# B&R Automation Studio project TD52 (part 150)

#### OpcMDE.st
```iecst
(*******************************************************************************
OPC_MDE	 Variables read or write to Measurement

This code is confidential AND proprietary to the INNIO Company.
It may NOT be used in any form, or reproduced in any manner, without the express
written permission of the INNIO Company.
Copyright, INNIO Company, 2022

- list addidtional customized IO channels

Customized modifications: -
------------------------

History:
-------
V1.00.0	09.12.2022		Vockenberger	Neu erstellt
V1.02.0	10.04.2024		Vockenberger	IN_DI.rP_Set auf IN_DI.rP_Act_FiltMDE + Mapping von MM2VIS.rP_Act_Filt
V1.03.0	05.03.2025		Vockenberger	added rOpcMDE_R[237] to rOpcMDE_R[300]

Instructions FOR use:
--------------------

Outstandings:
------------

*******************************************************************************)
PROGRAM _CYCLIC

	(*Connection OPC timeout*)
	(**BOOL**)
	TON_bComOpcBitMDE(IN:= bComOpcBitMDE, PT:=T#1s);
	IF TON_bComOpcBitMDE.Q THEN
		bOpcMDE_W[0] := FALSE;
	END_IF
	TON_bComOpcFailMDE(IN:= NOT bOpcMDE_W[0], PT:=T#1s);

	bComOpcBitMDE	:=	bOpcMDE_W[0];

	(*Abfrage welche Klopfüberwachung verwendet wird*)
	IF IN_DI.bKLS98_Active THEN
		rKnck_Sign[1] 	:= IN_DI.rKLS98_X_Window1[1];
		rKnck_Sign[2] 	:= IN_DI.rKLS98_X_Window1[2];
		rKnck_Sign[3] 	:= IN_DI.rKLS98_X_Window1[3];
		rKnck_Sign[4] 	:= IN_DI.rKLS98_X_Window1[4];
		rKnck_Sign[5] 	:= IN_DI.rKLS98_X_Window1[5];
		rKnck_Sign[6] 	:= IN_DI.rKLS98_X_Window1[6];
		rKnck_Sign[7] 	:= IN_DI.rKLS98_X_Window1[7];
		rKnck_Sign[8] 	:= IN_DI.rKLS98_X_Window1[8];
		rKnck_Sign[9] 	:= IN_DI.rKLS98_X_Window1[9];
		rKnck_Sign[10] 	:= IN_DI.rKLS98_X_Window1[10];
		rKnck_Sign[11] 	:= IN_DI.rKLS98_X_Window1[11];
		rKnck_Sign[12]	:= IN_DI.rKLS98_X_Window1[12];
		rKnck_Sign[13] 	:= IN_DI.rKLS98_X_Window1[13];
		rKnck_Sign[14] 	:= IN_DI.rKLS98_X_Window1[14];
		rKnck_Sign[15] 	:= IN_DI.rKLS98_X_Window1[15];
		rKnck_Sign[16] 	:= IN_DI.rKLS98_X_Window1[16];
		rKnck_Sign[17]	:= IN_DI.rKLS98_X_Window1[17];
		rKnck_Sign[18] 	:= IN_DI.rKLS98_X_Window1[18];
		rKnck_Sign[19] 	:= IN_DI.rKLS98_X_Window1[19];
		rKnck_Sign[20] 	:= IN_DI.rKLS98_X_Window1[20];
		rKnck_Sign[21] 	:= IN_DI.rKLS98_X_Window1[21];
		rKnck_Sign[22] 	:= IN_DI.rKLS98_X_Window1[22];
		rKnck_Sign[23] 	:= IN_DI.rKLS98_X_Window1[23];
		rKnck_Sign[24] 	:= IN_DI.rKLS98_X_Window1[24];
	ELSIF IN_DI.bSA_KLS_Active THEN
		rKnck_Sign[1] 	:= INT_TO_REAL(IN_DI.iU_SAFI_Win1[1]);
		rKnck_Sign[2] 	:= INT_TO_REAL(IN_DI.iU_SAFI_Win1[2]);
		rKnck_Sign[3] 	:= INT_TO_REAL(IN_DI.iU_SAFI_Win1[3]);
		rKnck_Sign[4] 	:= INT_TO_REAL(IN_DI.iU_SAFI_Win1[4]);
		rKnck_Sign[5] 	:= INT_TO_REAL(IN_DI.iU_SAFI_Win1[5]);
		rKnck_Sign[6] 	:= INT_TO_REAL(IN_DI.iU_SAFI_Win1[6]);
		rKnck_Sign[7] 	:= INT_TO_REAL(IN_DI.iU_SAFI_Win1[7]);
		rKnck_Sign[8] 	:= INT_TO_REAL(IN_DI.iU_SAFI_Win1[8]);
		rKnck_Sign[9] 	:= INT_TO_REAL(IN_DI.iU_SAFI_Win1[9]);
		rKnck_Sign[10] 	:= INT_TO_REAL(IN_DI.iU_SAFI_Win1[10]);
		rKnck_Sign[11] 	:= INT_TO_REAL(IN_DI.iU_SAFI_Win1[11]);
		rKnck_Sign[12]	:= INT_TO_REAL(IN_DI.iU_SAFI_Win1[12]);
		rKnck_Sign[13] 	:= INT_TO_REAL(IN_DI.iU_SAFI_Win1[13]);
		rKnck_Sign[14] 	:= INT_TO_REAL(IN_DI.iU_SAFI_Win1[14]);
		rKnck_Sign[15] 	:= INT_TO_REAL(IN_DI.iU_SAFI_Win1[15]);
		rKnck_Sign[16] 	:= INT_TO_REAL(IN_DI.iU_SAFI_Win1[16]);
		rKnck_Sign[17]	:= INT_TO_REAL(IN_DI.iU_SAFI_Win1[17]);
		rKnck_Sign[18] 	:= INT_TO_REAL(IN_DI.iU_SAFI_Win1[18]);
		rKnck_Sign[19] 	:= INT_TO_REAL(IN_DI.iU_SAFI_Win1[19]);
		rKnck_Sign[20] 	:= INT_TO_REAL(IN_DI.iU_SAFI_Win1[20]);
		rKnck_Sign[21] 	:= INT_TO_REAL(IN_DI.iU_SAFI_Win1[21]);
		rKnck_Sign[22] 	:= INT_TO_REAL(IN_DI.iU_SAFI_Win1[22]);
		rKnck_Sign[23] 	:= INT_TO_REAL(IN_DI.iU_SAFI_Win1[23]);
		rKnck_Sign[24] 	:= INT_TO_REAL(IN_DI.iU_SAFI_Win1[24]);
	ELSIF IN_DI.bSA_PI_Active THEN
		rKnck_Sign[1] 	:= IN_DI.rPr_Knck[1] * 1000;
		rKnck_Sign[2] 	:= IN_DI.rPr_Knck[2] * 1000;
		rKnck_Sign[3] 	:= IN_DI.rPr_Knck[3] * 1000;
		rKnck_Sign[4] 	:= IN_DI.rPr_Knck[4] * 1000;
		rKnck_Sign[5] 	:= IN_DI.rPr_Knck[5] * 1000;
		rKnck_Sign[6] 	:= IN_DI.rPr_Knck[6] * 1000;
		rKnck_Sign[7] 	:= IN_DI.rPr_Knck[7] * 1000;
		rKnck_Sign[8] 	:= IN_DI.rPr_Knck[8] * 1000;
		rKnck_Sign[9] 	:= IN_DI.rPr_Knck[9] * 1000;
		rKnck_Sign[10] 	:= IN_DI.rPr_Knck[10] * 1000;
		rKnck_Sign[11] 	:= IN_DI.rPr_Knck[11] * 1000;
		rKnck_Sign[12]	:= IN_DI.rPr_Knck[12] * 1000;
		rKnck_Sign[13] 	:= IN_DI.rPr_Knck[13] * 1000;
		rKnck_Sign[14] 	:= IN_DI.rPr_Knck[14] * 1000;
		rKnck_Sign[15] 	:= IN_DI.rPr_Knck[15] * 1000;
		rKnck_Sign[16] 	:= IN_DI.rPr_Knck[16] * 1000;
		rKnck_Sign[17]	:= IN_DI.rPr_Knck[17] * 1000;
		rKnck_Sign[18] 	:= IN_DI.rPr_Knck[18] * 1000;
		rKnck_Sign[19] 	:= IN_DI.rPr_Knck[19] * 1000;
		rKnck_Sign[20] 	:= IN_DI.rPr_Knck[20] * 1000;
		rKnck_Sign[21] 	:= IN_DI.rPr_Knck[21] * 1000;
		rKnck_Sign[22] 	:= IN_DI.rPr_Knck[22] * 1000;
		rKnck_Sign[23] 	:= IN_DI.rPr_Knck[23] * 1000;
		rKnck_Sign[24] 	:= IN_DI.rPr_Knck[24] * 1000;
	ELSE
		rKnck_Sign[1] 	:= 0;
		rKnck_Sign[2] 	:= 0;
		rKnck_Sign[3] 	:= 0;
		rKnck_Sign[4] 	:= 0;
		rKnck_Sign[5] 	:= 0;
		rKnck_Sign[6] 	:= 0;
		rKnck_Sign[7] 	:= 0;
		rKnck_Sign[8] 	:= 0;
		rKnck_Sign[9] 	:= 0;
		rKnck_Sign[10] 	:= 0;
		rKnck_Sign[11] 	:= 0;
		rKnck_Sign[12]	:= 0;
		rKnck_Sign[13] 	:= 0;
		rKnck_Sign[14] 	:= 0;
		rKnck_Sign[15] 	:= 0;
		rKnck_Sign[16] 	:= 0;
		rKnck_Sign[17]	:= 0;
		rKnck_Sign[18] 	:= 0;
		rKnck_Sign[19] 	:= 0;
		rKnck_Sign[20] 	:= 0;
		rKnck_Sign[21] 	:= 0;
		rKnck_Sign[22] 	:= 0;
		rKnck_Sign[23] 	:= 0;
		rKnck_Sign[24] 	:= 0;
	END_IF

	(*OPC Var to MDE*)
	rOpcMDE_R[0]	:=	DINT_TO_REAL(IN_DI.iCnt_OpHours);
	rOpcMDE_R[1]	:=	IN_DI.rT_EPU_EG[1];
	rOpcMDE_R[2]	:=	IN_DI.rT_EPU_EG[2];
	rOpcMDE_R[3]	:=	IN_DI.rT_EPU_EG[3];
	rOpcMDE_R[4]	:=	IN_DI.rT_EPU_EG[4];
	rOpcMDE_R[5]	:=	IN_DI.rT_EPU_EG[5];
	rOpcMDE_R[6]	:=	IN_DI.rT_EPU_EG[6];
	rOpcMDE_R[7]	:=	IN_DI.rT_EPU_EG[7];
	rOpcMDE_R[8]	:=	IN_DI.rT_EPU_EG[8];
	rOpcMDE_R[9]	:=	IN_DI.rT_EPU_EG[9];
	rOpcMDE_R[10]	:=	IN_DI.rT_EPU_EG[10];
	rOpcMDE_R[11]	:=	IN_DI.rT_EPU_EG[11];
	rOpcMDE_R[12]	:=	IN_DI.rT_EPU_EG[12];
	rOpcMDE_R[13]	:=	IN_DI.rT_EPU_EG[13];
	rOpcMDE_R[14]	:=	IN_DI.rT_EPU_EG[14];
	rOpcMDE_R[15]	:=	IN_DI.rT_EPU_EG[15];
	rOpcMDE_R[16]	:=	IN_DI.rT_EPU_EG[16];
	rOpcMDE_R[17]	:=	IN_DI.rT_EPU_EG[17];
	rOpcMDE_R[18]	:=	IN_DI.rT_EPU_EG[18];
	rOpcMDE_R[19]	:=	IN_DI.rT_EPU_EG[19];
	rOpcMDE_R[20]	:=	IN_DI.rT_EPU_EG[20];
	rOpcMDE_R[21]	:=	IN_DI.rT_EPU_EG[21];
	rOpcMDE_R[22]	:=	IN_DI.rT_EPU_EG[22];
	rOpcMDE_R[23]	:=	IN_DI.rT_EPU_EG[23];
	rOpcMDE_R[24]	:=	IN_DI.rT_EPU_EG[24];
	rOpcMDE_R[25]	:=	rKnck_Sign[1];
	rOpcMDE_R[26]	:=	rKnck_Sign[2];
	rOpcMDE_R[27]	:=	rKnck_Sign[3];
	rOpcMDE_R[28]	:=	rKnck_Sign[4];
	rOpcMDE_R[29]	:=	rKnck_Sign[5];
	rOpcMDE_R[30]	:=	rKnck_Sign[6];
	rOpcMDE_R[31]	:=	rKnck_Sign[7];
	rOpcMDE_R[32]	:=	rKnck_Sign[8];
	rOpcMDE_R[33]	:=	rKnck_Sign[9];
	rOpcMDE_R[34]	:=	rKnck_Sign[10];
	rOpcMDE_R[35]	:=	rKnck_Sign[11];
	rOpcMDE_R[36]	:=	rKnck_Sign[12];
	rOpcMDE_R[37]	:=	rKnck_Sign[13];
	rOpcMDE_R[38]	:=	rKnck_Sign[14];
	rOpcMDE_R[39]	:=	rKnck_Sign[15];
	rOpcMDE_R[40]	:=	rKnck_Sign[16];
	rOpcMDE_R[41]	:=	rKnck_Sign[17];
	rOpcMDE_R[42]	:=	rKnck_Sign[18];
	rOpcMDE_R[43]	:=	rKnck_Sign[19];
	rOpcMDE_R[44]	:=	rKnck_Sign[20];
	rOpcMDE_R[45]	:=	rKnck_Sign[21];
	rOpcMDE_R[46]	:=	rKnck_Sign[22];
	rOpcMDE_R[47]	:=	rKnck_Sign[23];
	rOpcMDE_R[48]	:=	rKnck_Sign[24];
	rOpcMDE_R[49]	:=	IN_DI.rCA_PI_Dur[1];
	rOpcMDE_R[50]	:=	IN_DI.rCA_PI_Dur[2];
	rOpcMDE_R[51]	:=	IN_DI.rCA_PI_Dur[3];
	rOpcMDE_R[52]	:=	IN_DI.rCA_PI_Dur[4];
	rOpcMDE_R[53]	:=	IN_DI.rCA_PI_Dur[5];
	rOpcMDE_R[54]	:=	IN_DI.rCA_PI_Dur[6];
	rOpcMDE_R[55]	:=	IN_DI.rCA_PI_Dur[7];
	rOpcMDE_R[56]	:=	IN_DI.rCA_PI_Dur[8];
	rOpcMDE_R[57]	:=	IN_DI.rCA_PI_Dur[9];
	rOpcMDE_R[58]	:=	IN_DI.rCA_PI_Dur[10];
	rOpcMDE_R[59]	:=	IN_DI.rCA_PI_Dur[11];
	rOpcMDE_R[60]	:=	IN_DI.rCA_PI_Dur[12];
	rOpcMDE_R[61]	:=	IN_DI.rCA_PI_Dur[13];
	rOpcMDE_R[62]	:=	IN_DI.rCA_PI_Dur[14];
	rOpcMDE_R[63]	:=	IN_DI.rCA_PI_Dur[15];
	rOpcMDE_R[64]	:=	IN_DI.rCA_PI_Dur[16];
	rOpcMDE_R[65]	:=	IN_DI.rCA_PI_Dur[17];
	rOpcMDE_R[66]	:=	IN_DI.rCA_PI_Dur[18];
	rOpcMDE_R[67]	:=	IN_DI.rCA_PI_Dur[19];
	rOpcMDE_R[68]	:=	IN_DI.rCA_PI_Dur[20];
	rOpcMDE_R[69]	:=	IN_DI.rCA_PI_Dur[21];
	rOpcMDE_R[70]	:=	IN_DI.rCA_PI_Dur[22];
	rOpcMDE_R[71]	:=	IN_DI.rCA_PI_Dur[23];
	rOpcMDE_R[72]	:=	IN_DI.rCA_PI_Dur[24];
	rOpcMDE_R[73]	:=	IN_DI.rCA_Ign_Act[1];
	rOpcMDE_R[74]	:=	IN_DI.rCA_Ign_Act[2];
	rOpcMDE_R[75]	:=	IN_DI.rCA_Ign_Act[3];
	rOpcMDE_R[76]	:=	IN_DI.rCA_Ign_Act[4];
	rOpcMDE_R[77]	:=	IN_DI.rCA_Ign_Act[5];
	rOpcMDE_R[78]	:=	IN_DI.rCA_Ign_Act[6];
	rOpcMDE_R[79]	:=	IN_DI.rCA_Ign_Act[7];
	rOpcMDE_R[80]	:=	IN_DI.rCA_Ign_Act[8];
	rOpcMDE_R[81]	:=	IN_DI.rCA_Ign_Act[9];
	rOpcMDE_R[82]	:=	IN_DI.rCA_Ign_Act[10];
	rOpcMDE_R[83]	:=	IN_DI.rCA_Ign_Act[11];
	rOpcMDE_R[84]	:=	IN_DI.rCA_Ign_Act[12];
	rOpcMDE_R[85]	:=	IN_DI.rCA_Ign_Act[13];
	rOpcMDE_R[86]	:=	IN_DI.rCA_Ign_Act[14];
	rOpcMDE_R[87]	:=	IN_DI.rCA_Ign_Act[15];
	rOpcMDE_R[88]	:=	IN_DI.rCA_Ign_Act[16];
	rOpcMDE_R[89]	:=	IN_DI.rCA_Ign_Act[17];
	rOpcMDE_R[90]	:=	IN_DI.rCA_Ign_Act[18];
	rOpcMDE_R[91]	:=	IN_DI.rCA_Ign_Act[19];
	rOpcMDE_R[92]	:=	IN_DI.rCA_Ign_Act[20];
	rOpcMDE_R[93]	:=	IN_DI.rCA_Ign_Act[21];
	rOpcMDE_R[94]	:=	IN_DI.rCA_Ign_Act[22];
	rOpcMDE_R[95]	:=	IN_DI.rCA_Ign_Act[23];
	rOpcMDE_R[96]	:=	IN_DI.rCA_Ign_Act[24];
	rOpcMDE_R[97]	:=	IN_DI.rU_Ign_Cyl[1];
	rOpcMDE_R[98]	:=	IN_DI.rU_Ign_Cyl[2];
	rOpcMDE_R[99]	:=	IN_DI.rU_Ign_Cyl[3];
	rOpcMDE_R[100]	:=	IN_DI.rU_Ign_Cyl[4];
	rOpcMDE_R[101]	:=	IN_DI.rU_Ign_Cyl[5];
	rOpcMDE_R[102]	:=	IN_DI.rU_Ign_Cyl[6];
	rOpcMDE_R[103]	:=	IN_DI.rU_Ign_Cyl[7];
	rOpcMDE_R[104]	:=	IN_DI.rU_Ign_Cyl[8];
	rOpcMDE_R[105]	:=	IN_DI.rU_Ign_Cyl[9];
	rOpcMDE_R[106]	:=	IN_DI.rU_Ign_Cyl[10];
	rOpcMDE_R[107]	:=	IN_DI.rU_Ign_Cyl[11];
	rOpcMDE_R[108]	:=	IN_DI.rU_Ign_Cyl[12];
	rOpcMDE_R[109]	:=	IN_DI.rU_Ign_Cyl[13];
	rOpcMDE_R[110]	:=	IN_DI.rU_Ign_Cyl[14];
	rOpcMDE_R[111]	:=	IN_DI.rU_Ign_Cyl[15];
	rOpcMDE_R[112]	:=	IN_DI.rU_Ign_Cyl[16];
	rOpcMDE_R[113]	:=	IN_DI.rU_Ign_Cyl[17];
	rOpcMDE_R[114]	:=	IN_DI.rU_Ign_Cyl[18];
	rOpcMDE_R[115]	:=	IN_DI.rU_Ign_Cyl[19];
	rOpcMDE_R[116]	:=	IN_DI.rU_Ign_Cyl[20];
	rOpcMDE_R[117]	:=	IN_DI.rU_Ign_Cyl[21];
	rOpcMDE_R[118]	:=	IN_DI.rU_Ign_Cyl[22];
	rOpcMDE_R[119]	:=	IN_DI.rU_Ign_Cyl[23];
	rOpcMDE_R[120]	:=	IN_DI.rU_Ign_Cyl[24];
	rOpcMDE_R[121]	:=	IN_DI.rT_CBearing[1];
	rOpcMDE_R[122]	:=	IN_DI.rT_CBearing[2];
	rOpcMDE_R[123]	:=	IN_DI.rT_CBearing[3];
	rOpcMDE_R[124]	:=	IN_DI.rT_CBearing[4];
	rOpcMDE_R[125]	:=	IN_DI.rT_CBearing[5];
	rOpcMDE_R[126]	:=	IN_DI.rT_CBearing[6];
	rOpcMDE_R[127]	:=	IN_DI.rT_CBearing[7];
	rOpcMDE_R[128]	:=	IN_DI.rT_CBearing[8];
	rOpcMDE_R[129]	:=	IN_DI.rT_CBearing[9];
	rOpcMDE_R[130]	:=	IN_DI.rT_CBearing[10];
	rOpcMDE_R[131]	:=	IN_DI.rT_CBearing[11];
	rOpcMDE_R[132]	:=	IN_DI.rT_CBearing[12];
	rOpcMDE_R[133]	:=	IN_DI.rT_CBearing[13];
	rOpcMDE_R[134]	:=	IN_DI.rT_CBearing[14];
	rOpcMDE_R[135]	:=	IN_DI.rT_CBearing[15];
	rOpcMDE_R[136]	:=	IN_DI.rT_CBearing[16];
	rOpcMDE_R[137]	:=	IN_DI.rT_CBearing[17];
	rOpcMDE_R[138]	:=	IN_DI.rT_CBearing[18];
	rOpcMDE_R[139]	:=	IN_DI.rT_CBearing[19];
	rOpcMDE_R[140]	:=	IN_DI.rT_CBearing[20];
	rOpcMDE_R[141]	:=	IN_DI.rT_CBearing[21];
	rOpcMDE_R[142]	:=	IN_DI.rT_CBearing[22];
	rOpcMDE_R[143]	:=	IN_DI.rT_CBearing[23];
	rOpcMDE_R[144]	:=	IN_DI.rT_CBearing[24];
	rOpcMDE_R[145]	:=	IN_DI.tT_MBearing[1].Ai;
	rOpcMDE_R[146]	:=	IN_DI.tT_MBearing[2].Ai;
	rOpcMDE_R[147]	:=	IN_DI.tT_MBearing[3].Ai;
	rOpcMDE_R[148]	:=	IN_DI.tT_MBearing[4].Ai;
	rOpcMDE_R[149]	:=	IN_DI.tT_MBearing[5].Ai;
	rOpcMDE_R[150]	:=	IN_DI.tT_MBearing[6].Ai;
	rOpcMDE_R[151]	:=	IN_DI.tT_MBearing[7].Ai;
	rOpcMDE_R[152]	:=	IN_DI.tT_MBearing[8].Ai;
	rOpcMDE_R[153]	:=	IN_DI.tT_MBearing[9].Ai;
	rOpcMDE_R[154]	:=	IN_DI.tT_MBearing[10].Ai;
	rOpcMDE_R[155]	:=	IN_DI.tT_MBearing[11].Ai;
	rOpcMDE_R[156]	:=	IN_DI.rCA_IgnP_Set;
	rOpcMDE_R[157]	:=	IN_DI.rCA_PI_Dur_Avg;
	rOpcMDE_R[158]	:=	IN_DI.rLam_Eng_LL_Set;
	rOpcMDE_R[159]	:=	IN_DI.rCA_Ign_Min;
	rOpcMDE_R[160]	:=	IN_DI.rCA_Ign_Max;
	rOpcMDE_R[161]	:=	IN_DI.rN_EngAct;
	IF IN_DI.tPos_Act_TV_A1.Exist THEN
		rOpcMDE_R[162]	:=	IN_DI.tPos_TV_A1.Ao;
	ELSE
		rOpcMDE_R[162]	:=	IN_DI.tPos_TV.Ao;
	END_IF
	rOpcMDE_R[163]	:=	IN_DI.rO2_NOxS_EngOut_B;
	rOpcMDE_R[164]	:=	IN_DI.tPos_TV_A2.Ao;
	rOpcMDE_R[165]	:=	IN_DI.tPos_TV_B1.Ao;
	rOpcMDE_R[166]	:=	IN_DI.tPos_TV_B2.Ao;
	IF IN_DI.bTSTC_Exist THEN
		rOpcMDE_R[167]	:=	IN_DI.tPos_CBV_A1.Ao;
		rOpcMDE_R[168]	:=	IN_DI.tPos_CBV_A2.Ao;
	ELSE
		rOpcMDE_R[167]	:=	IN_DI.tPos_CBV.Ao;
		rOpcMDE_R[168]	:=	IN_DI.tPos_CBV.Ao;
	END_IF
	rOpcMDE_R[169]	:=	IN_DI.rT_Ch_T2s_Avg;
	rOpcMDE_R[170]	:=	IN_DI.rCA_Ign_Avg;
	IF IN_DI.bTSTC_Exist THEN
		rOpcMDE_R[171]	:=	IN_DI.tPos_CBV_B1.Ao;
		rOpcMDE_R[172]	:=	IN_DI.tPos_CBV_B2.Ao;
	ELSE
		rOpcMDE_R[171]	:=	IN_DI.tPos_CBV34.Ao;
		rOpcMDE_R[172]	:=	IN_DI.tPos_CBV34.Ao;
	END_IF
	IF IN_DI.tPos_Act_TV_A1.Exist THEN
		rOpcMDE_R[173]	:=	IN_DI.tPos_Act_TV_A1.Ai;
	ELSE
		rOpcMDE_R[173]	:=	IN_DI.tPos_Act_TV.Ai;
	END_IF
	rOpcMDE_R[174]	:=	IN_DI.rO2_NOxS_EngOut;
	rOpcMDE_R[175]	:=	IN_DI.tPos_Act_TV_A2.Ai;
	rOpcMDE_R[176]	:=	IN_DI.tPos_Act_TV_B1.Ai;
	rOpcMDE_R[177]	:=	IN_DI.tPos_Act_TV_B2.Ai;
	IF IN_DI.tPos_Act_CBV_1.Exist THEN
		rOpcMDE_R[178]	:=	IN_DI.tPos_Act_CBV_1.Ai;
	ELSE
		rOpcMDE_R[178]	:=	IN_DI.tPos_Act_CBV_A1.Ai;
	END_IF
	IF IN_DI.tPos_Act_CBV_2.Exist THEN
		rOpcMDE_R[179]	:=	IN_DI.tPos_Act_CBV_2.Ai;
	ELSE
		rOpcMDE_R[179]	:=	IN_DI.tPos_Act_CBV_A2.Ai;
	END_IF
	IF IN_DI.tPos_Act_CBV_3.Exist THEN
		rOpcMDE_R[180]	:=	IN_DI.tPos_Act_CBV_3.Ai;
	ELSE
		rOpcMDE_R[180]	:=	IN_DI.tPos_Act_CBV_B1.Ai;
	END_IF
	rOpcMDE_R[181]	:=	IN_DI.tPos_Act_CBV_B2.Ai;
	rOpcMDE_R[182]	:=	UDINT_TO_REAL(IN_DI.ulGasFlowN[1]);
	rOpcMDE_R[183]	:=	UDINT_TO_REAL(IN_DI.ulGasFlowN[2]);
	rOpcMDE_R[184]	:=	UDINT_TO_REAL(IN_DI.ulGasFlowN[3]);
	rOpcMDE_R[185]	:=	IN_DI.rPr_EngLubOil;
	rOpcMDE_R[186]	:=	IN_DI.rT_EO;
	rOpcMDE_R[187]	:=	IN_DI.rT_ECW;
	rOpcMDE_R[188]	:=	IN_DI.rPr_ECW;
	rOpcMDE_R[189]	:=	IN_DI.rPr_TC_EOF_After;
	IF IN_DI.tPr_Ch_P2s_A.Exist THEN
		rOpcMDE_R[190]	:=	IN_DI.tPr_Ch_P2s_A.Ai;
	ELSE
		rOpcMDE_R[190]	:=	IN_DI.rPr_Ch_P2s;
	END_IF
	rOpcMDE_R[191]	:=	IN_DI.rO2_NOxS_EngOut_A;
	rOpcMDE_R[192]	:=	IN_DI.rPr_Ch_P2s_B;
	rOpcMDE_R[193]	:=	IN_DI.rPr_ECWaEng;
	rOpcMDE_R[194]	:=	IN_DI.rU_Avg_1;
	rOpcMDE_R[195]	:=	IN_DI.rI_Avg_1;
	rOpcMDE_R[196]	:=	IN_DI.rPF_Act_1;
	rOpcMDE_R[197]	:=	IN_DI.rPr_GR_I;
	rOpcMDE_R[198]	:=	IN_DI.rT_GR;
	rOpcMDE_R[199]	:=	IN_DI.rT_PCGT;
	rOpcMDE_R[200]	:=	IN_DI.rPr_PCG;
	rOpcMDE_R[201]	:=	IN_DI.rU_L1L2_1;
	rOpcMDE_R[202]	:=	IN_DI.rU_L2L3_1;
	rOpcMDE_R[203]	:=	IN_DI.rU_L3L1_1;
	rOpcMDE_R[204]	:=	IN_DI.rU_L1N_1;
	rOpcMDE_R[205]	:=	IN_DI.rU_L2N_1;
	rOpcMDE_R[206]	:=	IN_DI.rU_L3N_1;
	rOpcMDE_R[207]	:=	IN_DI.rPr_CC;
	rOpcMDE_R[208]	:=	IN_DI.rPr_EOF_DiffMon;
	rOpcMDE_R[209]	:=	IN_DI.rP_WorkAct_1;
	IF IN_DI.rNOx_NOxS_EngOut_Filt > 0.001 THEN
		rOpcMDE_R[210]	:=	IN_DI.rNOx_NOxS_EngOut_Filt;
	ELSE
		rOpcMDE_R[210]	:=	IN_DI.rNOx_NOxS_EngOut_A_Filt;
	END_IF
	rOpcMDE_R[211]	:=	IN_DI.rNOx_NOxS_EngOut_B_Filt;
	IF IN_DI.bN_TCHP_Exist THEN
		rOpcMDE_R[212]	:=	IN_DI.rN_TCHP;
	ELSE
		rOpcMDE_R[212]	:=	IN_DI.rN_TCHP_A;
	END_IF
	rOpcMDE_R[213]	:=	IN_DI.rN_TCHP_B;

	IF IN_DI.bN_TCHP_Exist THEN
		rOpcMDE_R[214]	:=	IN_DI.rN_TCLP;
	ELSE
		rOpcMDE_R[214]	:=	IN_DI.rN_TCLP_A;
	END_IF
	rOpcMDE_R[215]	:=	IN_DI.rN_TCLP_B;
	rOpcMDE_R[216]	:=	IN_DI.rGMU_Q_FuelGas[1];
	rOpcMDE_R[217]	:=	IN_DI.rGMU_Q_FuelGas[2];
	rOpcMDE_R[218]	:=	IN_DI.rGMU_Q_FuelGas[3];
	rOpcMDE_R[219]	:=	IN_DI.rGMU_Pos_Valve_Prom[1];
	rOpcMDE_R[220]	:=	IN_DI.rGMU_Pos_Valve_Prom[2];
	rOpcMDE_R[221]	:=	IN_DI.rGMU_Pos_Valve_Prom[3];
	rOpcMDE_R[222]	:=	IN_DI.rPr_PC_Diff;
	rOpcMDE_R[223]	:=	IN_DI.rOC_Consum_Avg;
	rOpcMDE_R[224]	:=	DINT_TO_REAL(IN_DI.iCnt_Starts);
	rOpcMDE_R[225]	:=	IN_DI.rP_Act_FiltMDE;
	rOpcMDE_R[226]	:=	IN_DI.rP_set_vis;
	rOpcMDE_R[227]	:=	IN_DI.rPr_EOaP;
	rOpcMDE_R[228]	:=	IN_DI.rT_Ch_T1LP;
	rOpcMDE_R[229]	:=	IN_DI.rPr_TC_EOF_Before;
	rOpcMDE_R[230]	:=	IN_DI.rPr_Ch_P2s_Avg;
	IF IN_DI.tPos_Act_WG.Exist THEN
		rOpcMDE_R[231]	:=	IN_DI.tPos_Act_WG.Ai;
		rOpcMDE_R[233]	:=	IN_DI.tPos_Set_WG.Ao;
	ELSE
		rOpcMDE_R[231]	:=	IN_DI.tPos_Act_WG_A.Ai;
		rOpcMDE_R[233]	:=	IN_DI.tPos_Set_WG_A.Ao;
	END_IF
	rOpcMDE_R[232]	:=	IN_DI.tPos_Act_WG_B.Ai;
	rOpcMDE_R[234]	:=	IN_DI.tPos_Set_WG_B.Ao;
	rOpcMDE_R[235]	:=	IN_DI.tT_ECWbEng.Ai;
	rOpcMDE_R[236]	:=	IN_DI.rT_Ch_T1HP_Avg;

	(*V1.03.0 Start*)
	rOpcMDE_R[237]	:=	IN_DI.rKnck_Intgr[1];
	rOpcMDE_R[238]	:=	IN_DI.rKnck_Intgr[2];
	rOpcMDE_R[239]	:=	IN_DI.rKnck_Intgr[3];
	rOpcMDE_R[240]	:=	IN_DI.rKnck_Intgr[4];
	rOpcMDE_R[241]	:=	IN_DI.rKnck_Intgr[5];
	rOpcMDE_R[242]	:=	IN_DI.rKnck_Intgr[6];
	rOpcMDE_R[243]	:=	IN_DI.rKnck_Intgr[7];
	rOpcMDE_R[244]	:=	IN_DI.rKnck_Intgr[8];
	rOpcMDE_R[245]	:=	IN_DI.rKnck_Intgr[9];
	rOpcMDE_R[246]	:=	IN_DI.rKnck_Intgr[10];
	rOpcMDE_R[247]	:=	IN_DI.rKnck_Intgr[11];
	rOpcMDE_R[248]	:=	IN_DI.rKnck_Intgr[12];
	rOpcMDE_R[249]	:=	IN_DI.rKnck_Intgr[13];
	rOpcMDE_R[250]	:=	IN_DI.rKnck_Intgr[14];
	rOpcMDE_R[251]	:=	IN_DI.rKnck_Intgr[15];
	rOpcMDE_R[252]	:=	IN_DI.rKnck_Intgr[16];
	rOpcMDE_R[253]	:=	IN_DI.rKnck_Intgr[17];
	rOpcMDE_R[254]	:=	IN_DI.rKnck_Intgr[18];
	rOpcMDE_R[255]	:=	IN_DI.rKnck_Intgr[19];
	rOpcMDE_R[256]	:=	IN_DI.rKnck_Intgr[20];
	rOpcMDE_R[257]	:=	IN_DI.rKnck_Intgr[21];
	rOpcMDE_R[258]	:=	IN_DI.rKnck_Intgr[22];
	rOpcMDE_R[259]	:=	IN_DI.rKnck_Intgr[23];
	rOpcMDE_R[260]	:=	IN_DI.rKnck_Intgr[24];
	rOpcMDE_R[261]	:=	IN_DI.rGen_T_In;
	rOpcMDE_R[262]	:=	IN_DI.rPr_Leanox_Dev;
	rOpcMDE_R[263]	:=	UINT_TO_REAL(usDurationPI_A);
	rOpcMDE_R[264]	:=	UINT_TO_REAL(usDurationPI_B);
	rOpcMDE_R[265]	:=	IN_DI.rPr_IMEP_Avg;
	rOpcMDE_R[266]	:=	IN_DI.rPr_CPP_Avg;
	rOpcMDE_R[267]	:=	IN_DI.rCA_MFBvar_Avg;
	rOpcMDE_R[268]	:=	IN_DI.rT_Ch_T2s_A;
	rOpcMDE_R[269]	:=	IN_DI.rT_Ch_T2s_B;
	rOpcMDE_R[270]	:=	IN_DI.rT_DAI;
	rOpcMDE_R[271]	:=	IN_DI.rPos_DAI_Set_A;
	rOpcMDE_R[272]	:=	IN_DI.rPos_DAI_Set_B;
	rOpcMDE_R[273]	:=	IN_DI.rPos_DAI_Act_A;
	rOpcMDE_R[274]	:=	IN_DI.rPos_DAI_Act_B;
	rOpcMDE_R[275]	:=	IN_DI.rFlow_Dem_DAI;
	rOpcMDE_R[276]	:=	IN_DI.rNOx_NOxS_CatOut_cor;
	rOpcMDE_R[277]	:=	IN_DI.rNOx_Em_AvgShortTerm;
	rOpcMDE_R[278]	:=	IN_DI.rFlow_SCR_UreaDosingOut;
	rOpcMDE_R[279]	:=	IN_DI.rT_SCR_UreaDosingUnit_Release;
	rOpcMDE_R[280]	:=	IN_DI.rNOx_Em_EngOut_mg_Set;
	rOpcMDE_R[281]	:=	IN_DI.rT_SCR_CatAvg;
	rOpcMDE_R[282]	:=	IN_DI.rO2_NOxS_CatOut;
	rOpcMDE_R[283]	:=	IN_DI.rHum_CatOut;
	rOpcMDE_R[284]	:=	IN_DI.rPr_GR_filt;
	rOpcMDE_R[285]	:=	IN_DI.rN_AirStarter;
	rOpcMDE_R[286]	:=	IN_DI.rBbBlower_y;
	rOpcMDE_R[287]	:=	IN_DI.rPr_MGT_a_Filt;
	rOpcMDE_R[288]	:=	IN_DI.rPr_PCGT_Out;
	rOpcMDE_R[289]	:=	IN_DI.rVol_Ch_Engine_Norm;
	rOpcMDE_R[290]	:=	IN_DI.rT_EG_LimMax;
	rOpcMDE_R[291]	:=	INT_TO_REAL(IN_DI.iNum_SkipCyl_Act);
	rOpcMDE_R[292]	:=	IN_DI.rFlow_OilSkid_DE;
	rOpcMDE_R[293]	:=	IN_DI.rFlow_OilSkid_NDE;
	rOpcMDE_R[294]	:=	IN_DI.tPIopenH[1].timing;
	rOpcMDE_R[295]	:=	IN_DI.rPr_AirStarter_Supply;
	rOpcMDE_R[296]	:=	IN_DI.rPos_AWG_Set_A;
	rOpcMDE_R[297]	:=	IN_DI.rPos_AWG_Set_B;
	rOpcMDE_R[298]	:=	IN_DI.rPos_AWG_Act_A;
	rOpcMDE_R[299]	:=	IN_DI.rPos_AWG_Act_B;
	rOpcMDE_R[300];
	(*V1.03.0 End*)

	rOpcMDE_R[301]	:=	IN_DI.rCust_ME[1];
	rOpcMDE_R[302]	:=	IN_DI.rCust_ME[2];
	rOpcMDE_R[303]	:=	IN_DI.rCust_ME[3];
	rOpcMDE_R[304]	:=	IN_DI.rCust_ME[4];
	rOpcMDE_R[305]	:=	IN_DI.rCust_ME[5];
	rOpcMDE_R[306]	:=	IN_DI.rCust_ME[6];
	rOpcMDE_R[307]	:=	IN_DI.rCust_ME[7];
	rOpcMDE_R[308]	:=	IN_DI.rCust_ME[8];
	rOpcMDE_R[309]	:=	IN_DI.rCust_ME[9];
	rOpcMDE_R[310]	:=	IN_DI.rCust_ME[10];
	rOpcMDE_R[311]	:=	IN_DI.rCust_ME[11];
	rOpcMDE_R[312]	:=	IN_DI.rCust_ME[12];
	rOpcMDE_R[313]	:=	IN_DI.rCust_ME[13];
	rOpcMDE_R[314]	:=	IN_DI.rCust_ME[14];
	rOpcMDE_R[315]	:=	IN_DI.rCust_ME[15];
	rOpcMDE_R[316]	:=	IN_DI.rCust_ME[16];
	rOpcMDE_R[317]	:=	IN_DI.rCust_ME[17];
	rOpcMDE_R[318]	:=	IN_DI.rCust_ME[18];
	rOpcMDE_R[319]	:=	IN_DI.rCust_ME[19];
	rOpcMDE_R[320]	:=	IN_DI.rCust_ME[20];
	rOpcMDE_R[321]	:=	IN_DI.rCust_ME[21];
	rOpcMDE_R[322]	:=	IN_DI.rCust_ME[22];
	rOpcMDE_R[323]	:=	IN_DI.rCust_ME[23];
	rOpcMDE_R[324]	:=	IN_DI.rCust_ME[24];
	rOpcMDE_R[325]	:=	IN_DI.rCust_ME[25];
	rOpcMDE_R[326]	:=	IN_DI.rCust_ME[26];
	rOpcMDE_R[327]	:=	IN_DI.rCust_ME[27];
	rOpcMDE_R[328]	:=	IN_DI.rCust_ME[28];
	rOpcMDE_R[329]	:=	IN_DI.rCust_ME[29];
	rOpcMDE_R[330]	:=	IN_DI.rCust_ME[30];
	rOpcMDE_R[331]	:=	IN_DI.rCust_ME[31];
	rOpcMDE_R[332]	:=	IN_DI.rCust_ME[32];
	rOpcMDE_R[333]	:=	IN_DI.rCust_ME[33];
	rOpcMDE_R[334]	:=	IN_DI.rCust_ME[34];
	rOpcMDE_R[335]	:=	IN_DI.rCust_ME[35];
	rOpcMDE_R[336]	:=	IN_DI.rCust_ME[36];
	rOpcMDE_R[337]	:=	IN_DI.rCust_ME[37];
	rOpcMDE_R[338]	:=	IN_DI.rCust_ME[38];
	rOpcMDE_R[339]	:=	IN_DI.rCust_ME[39];
	rOpcMDE_R[340]	:=	IN_DI.rCust_ME[40];
	rOpcMDE_R[341]	:=	IN_DI.rCust_ME[41];
	rOpcMDE_R[342]	:=	IN_DI.rCust_ME[42];
	rOpcMDE_R[343]	:=	IN_DI.rCust_ME[43];
	rOpcMDE_R[344]	:=	IN_DI.rCust_ME[44];
	rOpcMDE_R[345]	:=	IN_DI.rCust_ME[45];
	rOpcMDE_R[346]	:=	IN_DI.rCust_ME[46];
	rOpcMDE_R[347]	:=	IN_DI.rCust_ME[47];
	rOpcMDE_R[348]	:=	IN_DI.rCust_ME[48];
	rOpcMDE_R[349]	:=	IN_DI.rCust_ME[49];
	rOpcMDE_R[350]	:=	IN_DI.rCust_ME[50];
	rOpcMDE_R[351]	:=	IN_DI.rCust_ME[51];
	rOpcMDE_R[352]	:=	IN_DI.rCust_ME[52];
	rOpcMDE_R[353]	:=	IN_DI.rCust_ME[53];
	rOpcMDE_R[354]	:=	IN_DI.rCust_ME[54];
	rOpcMDE_R[355]	:=	IN_DI.rCust_ME[55];
	rOpcMDE_R[356]	:=	IN_DI.rCust_ME[56];
	rOpcMDE_R[357]	:=	IN_DI.rCust_ME[57];
	rOpcMDE_R[358]	:=	IN_DI.rCust_ME[58];
	rOpcMDE_R[359]	:=	IN_DI.rCust_ME[59];
	rOpcMDE_R[360]	:=	IN_DI.rCust_ME[60];
	rOpcMDE_R[361]	:=	IN_DI.rCust_ME[61];
	rOpcMDE_R[362]	:=	IN_DI.rCust_ME[62];
	rOpcMDE_R[363]	:=	IN_DI.rCust_ME[63];
	rOpcMDE_R[364]	:=	IN_DI.rCust_ME[64];
	rOpcMDE_R[365]	:=	IN_DI.rCust_ME[65];
	rOpcMDE_R[366]	:=	IN_DI.rCust_ME[66];
	rOpcMDE_R[367]	:=	IN_DI.rCust_ME[67];
	rOpcMDE_R[368]	:=	IN_DI.rCust_ME[68];
	rOpcMDE_R[369]	:=	IN_DI.rCust_ME[69];
	rOpcMDE_R[370]	:=	IN_DI.rCust_ME[70];
	rOpcMDE_R[371]	:=	IN_DI.rCust_ME[71];
	rOpcMDE_R[372]	:=	IN_DI.rCust_ME[72];
	rOpcMDE_R[373]	:=	IN_DI.rCust_ME[73];
	rOpcMDE_R[374]	:=	IN_DI.rCust_ME[74];
	rOpcMDE_R[375]	:=	IN_DI.rCust_ME[75];
	rOpcMDE_R[376]	:=	IN_DI.rCust_ME[76];
	rOpcMDE_R[377]	:=	IN_DI.rCust_ME[77];
	rOpcMDE_R[378]	:=	IN_DI.rCust_ME[78];
	rOpcMDE_R[379]	:=	IN_DI.rCust_ME[79];
	rOpcMDE_R[380]	:=	IN_DI.rCust_ME[80];
	rOpcMDE_R[381]	:=	IN_DI.rCust_ME[81];
	rOpcMDE_R[382]	:=	IN_DI.rCust_ME[82];
	rOpcMDE_R[383]	:=	IN_DI.rCust_ME[83];
	rOpcMDE_R[384]	:=	IN_DI.rCust_ME[84];
	rOpcMDE_R[385]	:=	IN_DI.rCust_ME[85];
	rOpcMDE_R[386]	:=	IN_DI.rCust_ME[86];
	rOpcMDE_R[387]	:=	IN_DI.rCust_ME[87];
	rOpcMDE_R[388]	:=	IN_DI.rCust_ME[88];
	rOpcMDE_R[389]	:=	IN_DI.rCust_ME[89];
	rOpcMDE_R[390]	:=	IN_DI.rCust_ME[90];
	rOpcMDE_R[391]	:=	IN_DI.rCust_ME[91];
	rOpcMDE_R[392]	:=	IN_DI.rCust_ME[92];
	rOpcMDE_R[393]	:=	IN_DI.rCust_ME[93];
	rOpcMDE_R[394]	:=	IN_DI.rCust_ME[94];
	rOpcMDE_R[395]	:=	IN_DI.rCust_ME[95];
	rOpcMDE_R[396]	:=	IN_DI.rCust_ME[96];
	rOpcMDE_R[397]	:=	IN_DI.rCust_ME[97];
	rOpcMDE_R[398]	:=	IN_DI.rCust_ME[98];
	rOpcMDE_R[399]	:=	IN_DI.rCust_ME[99];
	rOpcMDE_R[400]	:=	IN_DI.rCust_ME[100];
	rOpcMDE_R[401]	:=	IN_DI.rCust_ME[101];
	rOpcMDE_R[402]	:=	IN_DI.rCust_ME[102];
	rOpcMDE_R[403]	:=	IN_DI.rCust_ME[103];
	rOpcMDE_R[404]	:=	IN_DI.rCust_ME[104];
	rOpcMDE_R[405]	:=	IN_DI.rCust_ME[105];
	rOpcMDE_R[406]	:=	IN_DI.rCust_ME[106];
	rOpcMDE_R[407]	:=	IN_DI.rCust_ME[107];
	rOpcMDE_R[408]	:=	IN_DI.rCust_ME[108];
	rOpcMDE_R[409]	:=	IN_DI.rCust_ME[109];
	rOpcMDE_R[410]	:=	IN_DI.rCust_ME[110];
	rOpcMDE_R[411]	:=	IN_DI.rCust_ME[111];
	rOpcMDE_R[412]	:=	IN_DI.rCust_ME[112];
	rOpcMDE_R[413]	:=	IN_DI.rCust_ME[113];
	rOpcMDE_R[414]	:=	IN_DI.rCust_ME[114];
	rOpcMDE_R[415]	:=	IN_DI.rCust_ME[115];
	rOpcMDE_R[416]	:=	IN_DI.rCust_ME[116];
	rOpcMDE_R[417]	:=	IN_DI.rCust_ME[117];
	rOpcMDE_R[418]	:=	IN_DI.rCust_ME[118];
	rOpcMDE_R[419]	:=	IN_DI.rCust_ME[119];
	rOpcMDE_R[420]	:=	IN_DI.rCust_ME[120];

	rOpcMDE_R[421]	:=	IN_DI.rCust_ME_10ms[1];
	rOpcMDE_R[422]	:=	IN_DI.rCust_ME_10ms[2];
	rOpcMDE_R[423]	:=	IN_DI.rCust_ME_10ms[3];
	rOpcMDE_R[424]	:=	IN_DI.rCust_ME_10ms[4];
	rOpcMDE_R[425]	:=	IN_DI.rCust_ME_10ms[5];
	rOpcMDE_R[426]	:=	IN_DI.rCust_ME_10ms[6];
	rOpcMDE_R[427]	:=	IN_DI.rCust_ME_10ms[7];
	rOpcMDE_R[428]	:=	IN_DI.rCust_ME_10ms[8];
	rOpcMDE_R[429]	:=	IN_DI.rCust_ME_10ms[9];
	rOpcMDE_R[430]	:=	IN_DI.rCust_ME_10ms[10];
	rOpcMDE_R[431]	:=	IN_DI.rCust_ME_10ms[11];
	rOpcMDE_R[432]	:=	IN_DI.rCust_ME_10ms[12];
	rOpcMDE_R[433]	:=	IN_DI.rCust_ME_10ms[13];
	rOpcMDE_R[434]	:=	IN_DI.rCust_ME_10ms[14];
	rOpcMDE_R[435]	:=	IN_DI.rCust_ME_10ms[15];
	rOpcMDE_R[436]	:=	IN_DI.rCust_ME_10ms[16];
	rOpcMDE_R[437]	:=	IN_DI.rCust_ME_10ms[17];
	rOpcMDE_R[438]	:=	IN_DI.rCust_ME_10ms[18];
	rOpcMDE_R[439]	:=	IN_DI.rCust_ME_10ms[19];
	rOpcMDE_R[440]	:=	IN_DI.rCust_ME_10ms[20];

	bOpcMDE_R[0]	:=	IN_DI.bEOP1DC_Dem;
	(*V1.03.0 Start*)
	bOpcMDE_R[1]	:=	IN_DI.bEng_Start;
	bOpcMDE_R[2]	:=	IN_DI.bEng_Dem_Aut;
	bOpcMDE_R[3]	:=	IN_DI.bGCB_On;
	bOpcMDE_R[4]	:=	IN_DI.bAirST_ValEngage;
	bOpcMDE_R[5]	:=	IN_DI.bAirST_ValStart;
	bOpcMDE_R[6]	:=	IN_DI.bTCOV_CoClose;
	bOpcMDE_R[7]	:=	IN_DI.bScavVaFailure;
	bOpcMDE_R[8]	:=	IN_DI.bEng_Dem;
	bOpcMDE_R[9]	:=	IN_DI.bChargeOff_Dem;
	(*V1.03.0 End*)

	rOpcMDE_W;
	OUT_DI.rCust_From_PUMA[1]	:=	rOpcMDE_W[25];
	OUT_DI.rCust_From_PUMA[2]	:=	rOpcMDE_W[26];
	OUT_DI.rCust_From_PUMA[3]	:=	rOpcMDE_W[27];
	OUT_DI.rCust_From_PUMA[4]	:=	rOpcMDE_W[28];
	OUT_DI.rCust_From_PUMA[5]	:=	rOpcMDE_W[29];
	OUT_DI.rCust_From_PUMA[6]	:=	rOpcMDE_W[30];
	OUT_DI.rCust_From_PUMA[7]	:=	rOpcMDE_W[31];
	OUT_DI.rCust_From_PUMA[8]	:=	rOpcMDE_W[32];
	OUT_DI.rCust_From_PUMA[9]	:=	rOpcMDE_W[33];
	OUT_DI.rCust_From_PUMA[10]	:=	rOpcMDE_W[34];
	OUT_DI.rCust_From_PUMA[11]	:=	rOpcMDE_W[35];
	OUT_DI.rCust_From_PUMA[12]	:=	rOpcMDE_W[36];

	OUT_DI.rAMA_CH4_ppm		:=	rOpcMDE_W[41];
	OUT_DI.rAMA_THC_ppm		:=	rOpcMDE_W[42];
	OUT_DI.rAMA_CO_ppm		:=	rOpcMDE_W[43];
	OUT_DI.rAMA_CO2_per		:=	rOpcMDE_W[44];
	OUT_DI.rAMA_O2_per		:=	rOpcMDE_W[45];
	OUT_DI.rAMA_NO_ppm		:=	rOpcMDE_W[46];
	OUT_DI.rAMA_NOx_ppm		:=	rOpcMDE_W[47];
	OUT_DI.rAMA_Status		:=	rOpcMDE_W[48];
	rOpcMDE_W[49];
	rOpcMDE_W[50];

	bOpcMDE_W;

END_PROGRAM
```

#### OpcMDE.var
```iecst
VAR
	rKnck_Sign : ARRAY[0..24]OF REAL; (* Cylinder Knocking Value/Pressure *)
END_VAR
```

### Program Logical/DataInterface/IN_DI (IEC) - Var from Customiezd Modul

#### IN_DI.st
```iecst
(*******************************************************************************
IN_DI	Variables from other modules

This code is confidential AND proprietary to the INNIO Company.
It may NOT be used in any form, or reproduced in any manner, without the express
written permission of the INNIO Company.
Copyright, INNIO Company, 2022

- list addidtional customized IO channels

Customized modifications: -
------------------------

History:
-------
V1.01.0	31.07.2023		Vockenberger	Neu erstellt
		04.03.2024		Gruber St.		changed connection for gasvalves visualization
V1.01.1	19.03.2024		Gruber St.		changed connection for gas proportioning valves
										moved vis mixgas ratio to Gnl_GT
		27.03.2024		Gruber St. 		added H2-Sensor engine

Instructions FOR use:
--------------------

Outstandings:
------------

*******************************************************************************)
PROGRAM _CYCLIC

	(*Variablen die von anderen Modulen kommen*)
	IN_DI.rP_Act_Norm_Filt;
	MM2VIS.bBlocGasMixButton := IN_DI.bEng_Aux_Dem_CDR;
	MM2VIS.bPCG_GV_Open := IN_DI.bPCG_GV_Open;
	MM2VIS.bGV1_Open := IN_DI.bGV1_Open;
	MM2VIS.bGV2_Open := IN_DI.bGV2_Open; // AND MM2VIS.bDem_GV_PG AND NOT MM2VIS.bGV3_Open;
	MM2VIS.bGV3_Open := IN_DI.bGV3_Open; // AND MM2VIS.bDem_GV_SG AND NOT Para.bSG_MFC_Used AND NOT MM2VIS.bDem_GV_PG;
	MM2VIS.bEng_Run := IN_DI.bEng_Run;
	MM2VIS.rLam_Eng_LL_Set := IN_DI.rLam_Eng_LL_Set;
	MM2VIS.rGMU_Pos_Valve_Prom1 := IN_DI.rGMU_Pos_Valve_Prom[1];
	MM2VIS.rGMU_Pos_Valve_Prom2 := IN_DI.rGMU_Pos_Valve_Prom[2];
	MM2VIS.rGMU_Pos_Valve_Prom3 := IN_DI.rGMU_Pos_Valve_Prom[3];
	MM2VIS.iIdx_SelGasTyp	:= IN_DI.iIdx_SelGasTyp;
	MM2VIS.iIdx_Gtyp_Act	:= IN_DI.iIdx_Gtyp_Act;
	MM2VIS.rPr_Ch_P2s_Avg	:= IN_DI.rPr_Ch_P2s_Avg;
	MM2VIS.rCA_IgnP_Set	:=	IN_DI.rCA_IgnP_Set;
	MM2VIS.bGEN2_preM_Act	:=	IN_DI.bGEN2_preM_Act;
	MM2VIS.rGT_H2	:= IN_DI.rCust_ME[5] * 0.1;	// IN_DI.rGT_H2 * 100;
	MM2VIS.rCA_Ign_Avg		:=	IN_DI.rCA_Ign_Avg;
END_PROGRAM
```

### Program Logical/DataInterface/OUT_DI (IEC) - Var to Customiezd Modul

#### OUT_DI.st
```iecst
(*******************************************************************************
OUT_DI	Variables to other modules

This code is confidential AND proprietary to the INNIO Company.
It may NOT be used in any form, or reproduced in any manner, without the express
written permission of the INNIO Company.
Copyright, INNIO Company, 2022

- list addidtional customized IO channels

Customized modifications: -
------------------------

History:
-------
V1.00.0	14.09.2022		Vockenberger	Neu erstellt
V1.01.0 17.07.2023		Gruber St.		added setpoint for gasmixing with gas proportioning valve
		07.08.2023		Vockenberger	Ext Vorgaben von MDE/MyPlant
		04.03.2024		Gruber St.		added setpoints for admixing special gas with gas proportioning valve
V1.01.1 13.03.2024		Gruber St.		added variables for admixing H2

Instructions FOR use:
--------------------

Outstandings:
------------

*******************************************************************************)
PROGRAM _CYCLIC

	(*Aktivierung Vorwärmung, wenn Betriebswahlschalter auf aus ist *)
	IF EDGEPOS(MM2VIS.bPreHeatWDay_On) THEN	(*Aktivierung Vorwärmung vom Prüfstand über eine positiven Flanke*)
		VIS2MM.bECW_PreH_Dem_Customized := TRUE;
	ELSE
		VIS2MM.bECW_PreH_Dem_Customized := VIS2MM.bECW_PreH_Dem_Customized;
	END_IF

	OUT_DI.bECW_PreH_Dem_Customized := VIS2MM.bECW_PreH_Dem_Customized; (*Aktivierung Vorwärmung Prüfstandsseitig, wird im General_Di nochmal beschrieben*)

	(*Ext P-Vorgabe, kann über PUMA/MyPlant vorgegeben werden*)
	IF NOT MM2VIS.bMsg7000 AND VIS2MM.iSelExtP_OPC_Set = 1 THEN
		OUT_DI.bOPC_Dem := MM2VIS.bOPC_Dem;
		OUT_DI.rP_OPC_Set := MM2VIS.rP_OPC_Set;
	ELSIF VIS2MM.iSelExtP_OPC_Set = 2 THEN
		OUT_DI.rP_OPC_Set := MM2VIS.rP_OPC_Set;
		OUT_DI.bOPC_Dem := MM2VIS.bOPC_Dem;
	ELSE
		OUT_DI.rP_OPC_Set := 0.5;
		OUT_DI.bOPC_Dem := FALSE;
	END_IF
	OUT_DI.bBusAlive := MM2VIS.bBusAlive;

	(*Ext Vorgaben von MDE*)
	OUT_DI.rCA_IgnP_CylOffset			:= MM2VIS.rCA_IgnP_CylOffset;
	OUT_DI.bLeanox_Man_Cust				:= MM2VIS.bLeanox_Man_Cust;
	OUT_DI.rLam_Eng_LL_ManSet_Cust		:= MM2VIS.rLam_Eng_LL_ManSet_Cust;
	OUT_DI.rPr_Leanox_ManSet_Cust		:= MM2VIS.rPr_Leanox_ManSet_Cust;
	OUT_DI.bCA_IgnP_CylOffset_Active	:= MM2VIS.bCA_IgnP_CylOffset_Active;
	OUT_DI.bExtNOX_Active				:= MM2VIS.bExtNOX_Active;
	OUT_DI.rNOX_ManSet_Cust				:= MM2VIS.rNOX_ManSet_Cust;

	(*Gasmischen*)
	OUT_DI.bGT_CalibrateActive_Bus;
	OUT_DI.bCV_Bus_Active 		:= MM2VIS.bCV_Bus_Active;
	OUT_DI.rCV_Bus 				:= MM2VIS.rGT_CV_TB;
	OUT_DI.bOptGT_RatioMix_Set 	:= MM2VIS.bOptGT_RatioMix_Set;
	OUT_DI.rGT_RatioMix_Set		:= MM2VIS.rGT_RatioMix_Set;
	OUT_DI.bDem_GT3 			:= bDem_GT3;
	OUT_DI.rGT_RatioAdd			:= rGT_RatioAdd;
	OUT_DI.rH2_Set				:= rH2_Set;
	OUT_DI.rH2_Act_Calc			:= rH2_Act_Calc;
	OUT_DI.rH2_Act_Cube			:= rH2_Act_Cube;

END_PROGRAM
```

### Program Logical/DataInterface/PermDI (IEC, version 4.04.0) - + PermanentMemory

#### PermDICyclic.st - Cyclic code
```iecst
(*******************************************************************************
AGGR: read and write DIA.NE XT parameter to flash memory	(Cyclic)

This code is confidential and proprietary to the INNIO Jenbacher Company.
It may not be used in any form, or reproduced in any manner, without the express
written permission of the INNIO Company.
Copyright, INNIO Jenbacher Company, 2022

- every 10 seconds or at write once the parameter values are copied to the structure pm
- every 10 seconds the checksum of the parameter structure is calculate
- IF checksum has changed or write once is set the structure pm is written to
	the permanent memory data module

Customized modifications: -
------------------------

History:
-------
V1.00.0	16.09.2022	Vockenberger 	Neu erstellt
V1.01.0 07.08.2023	Vockenberger	im INIT Datenspeichergeändert, da neue Parameter dazukommen sind
V1.02.1 30.10.2024	Vockenberger	im INIT Datenspeichergeändert, da neue Parameter dazukommen sind

*******************************************************************************)
PROGRAM _CYCLIC

	(* 10 seconds timer *)
	TON_WritePMEM(IN := NOT TON_WritePMEM.Q, PT:= T#10s);
	TON_BlockMinFileAge(IN := bBlock_MinFileAge, PT:= T#10m);
	IF TON_BlockMinFileAge.Q  THEN bBlock_MinFileAge := FALSE; END_IF

	(* every 10 seconds or at write once the parameter values are copied to the structure pm *)
	IF TON_WritePMEM.Q OR write_once THEN

		(* ------------- V04.04.0 ---------------- *)   					(* permanent memory data *)
		pmm			:=	Para;						(* op.hours oxi cat *)

	END_IF;

	(* cyclic calcualtion of parameter checksum	*)
	IF TON_WritePMEM.Q THEN
		ulChecksum := 0;

		FOR ulPMPointer := ADR(pmm) TO (ADR(pmm) + pm_len - SIZEOF(ulChkValue)) DO
			memcpy(ADR(ulChkValue), ulPMPointer, SIZEOF(ulChkValue));
			ulChecksum := (ulChecksum XOR ulChkValue)+ulChkValue;
		END_FOR;

		IF ulChecksumOld <> ulChecksum THEN	(* if checksum has changed 		*)
			ulChecksumOld := ulChecksum;	(* save last cheksum value		*)
			bWriteDataObj := TRUE;			(* set flag for write checksum	*)
		END_IF;

	END_IF

	(* write structure pm to the permanent memory module *)
	IF ((bWriteDataObj AND NOT bBlock_MinFileAge) OR write_once) THEN

		DatObjWrite_01();									(* run data object write fub 				*)

		IF DatObjWrite_01.status <> ERR_FUB_BUSY THEN		(* wait if data object write fub is busy 	*)
			bWriteDataObj 	:= FALSE;						(* reset data object write flag				*)
			write_once 		:= FALSE;						(* reset write_once flag 					*)
			iPM_WriteCnt 	:= iPM_WriteCnt + 1;			(* counter for done data object module writes *)

			IF DatObjWrite_01.status = ERR_NOERROR THEN		(* if status = NO ERROR -> block further write requests for 10min to avoid CF wear down	*)
				bBlock_MinFileAge := TRUE;
			ELSE
				pm_Error := 2005;							(* set data object write error state		*)
			END_IF;
		END_IF;

	END_IF;

END_PROGRAM
```

#### PermDIInit.st - Initialization code
```iecst
(*******************************************************************************
AGGR: read and write DIA.NE XT parameter to flash memory	(init)

This code is confidential and proprietary to the INNIO Jenbacher Company.
It may not be used in any form, or reproduced in any manner, without the express
written permission of the INNIO Company.
Copyright, INNIO Jenbacher Company, 2022

- every 10 seconds or at write once the parameter values are copied to the structure pm
- every 10 seconds the checksum of the parameter structure is calculate
- IF checksum has changed or write once is set the structure pm is written to
	the permanent memory data module

Customized modifications: -
------------------------

History:
-------
V1.00.0	16.09.2022	Vockenberger 	Neu erstellt
V1.01.0 07.08.2023	Vockenberger	Datenspeichergeändert, da neue Parameter dazukommen sind
V1.01.1	20.03.2024	Gruber St.		Datenspeicher erhöht
V1.02.0 10.04.2024	Vockenberger	Datenspeichergeändert, da neue Parameter dazukommen sind
		23.04.2024	Gruber St.		Datenspeicher erhöht
V1.02.1 30.10.2024	Vockenberger	im INIT Datenspeichergeändert, da neue Parameter dazukommen sind

*******************************************************************************)

PROGRAM _INIT

	(* set some init parameters *)
	TON_WritePMEM(IN := FALSE, PT:= T#10s);			(* reset used timer function blocks 			*)

	pm_Error 	:= ERR_NOERROR;						(* reset permanent memory error	status			*)
	write_once 	:= FALSE;				 			(* reset flag for write permanent memory once	*)
	pm_len 		:= SIZEOF(pmm);						(* define data length of permenent memory		*)
	strcpy(ADR(ModulName),ADR('DataInterface::perm_DI'));	(* define name of permanent memory data module	*)

	(* check for existing permanent memory data module	*)
	DatObjInfo_01.enable:= TRUE;					(* enable FUB									*)
	DatObjInfo_01.pName := ADR(ModulName);			(* set permanent memory data module name 		*)
	DatObjInfo_01();								(* run data object info FUB						*)

	(* check error status of data object info FUB	*)
	IF DatObjInfo_01.status = ERR_NOERROR THEN		(* if no error	--> permanent memory data module exists	*)
		pm_id 	:= DatObjInfo_01.ident;				(* copy permanent memory data module ident			*)
		pm_p 	:= DatObjInfo_01.pDatObjMem;		(* copy permanent memory data module memory adres	*)
	ELSE
		bCreateDataObj := TRUE;						(* set flag for create new data object	*)
		pm_Error := 2001;							(* set permanent memory error status	*)
	END_IF;

	(* check length of parameter struct with length of data object *)

	CASE DatObjInfo_01.len OF

		1932: 		perm_par_vers  := 400;			(* 44 = length of perm_par V04.00.0 *)

			(* insert new perm_par Version here
			(* 		  bCreateDataObj := TRUE;		(* set flag for create new data object	*)
			(* xxxx:  perm_par_vers  := yyy;		(* xxxx = length of perm_par Vy.yy *)

		ELSE
		bCreateDataObj := TRUE;						(* set flag for create new data object	*)
	END_CASE;

	(* if permanent memory data module exist read data and copy to structure pm	*)
	IF pm_Error = ERR_NOERROR THEN					(* permanent memory data module exist 				*)
		DatObjRead_01.enable 		:= TRUE;		(* enable read permanent memory module data 		*)
		DatObjRead_01.ident 		:= pm_id;		(* set identifier of permanent memory data module	*)
		DatObjRead_01.Offset 		:= 0;			(* start at memory offest zero 						*)
		DatObjRead_01.pDestination := ADR(pmm);		(* set permanent data destination adress			*)
		DatObjRead_01.len 			:= DatObjInfo_01.len;	(* set length of permanent data module		*)

		REPEAT	(* repeat until data of permanent memory data module have been read *)
			DatObjRead_01();						(* FUB read data from permanent data module 		*)
			UNTIL	DatObjRead_01.status <> ERR_FUB_BUSY		(* wait if FUB is busy 	*)
		END_REPEAT;

		IF DatObjRead_01.status <> ERR_NOERROR THEN	(* if status of read permanent data moduel is not OK 	*)
			pm_Error :=2002;						(* set permanent memory error status					*)
		END_IF
	END_IF;

	IF NOT bCreateDataObj THEN
		(* if permanent memory data module exist read data and copy to structure pm	*)
		IF pm_Error = ERR_NOERROR THEN					(* permanent memory data module exist 				*)
			DatObjRead_01.enable 		:= TRUE;		(* enable read permanent memory module data 		*)
			DatObjRead_01.ident 		:= pm_id;		(* set identifier of permanent memory data module	*)
			DatObjRead_01.Offset 		:= 0;			(* start at memory offest zero 						*)
			DatObjRead_01.pDestination := ADR(pmm);		(* set permanent data destination adress			*)
			DatObjRead_01.len 			:= DatObjInfo_01.len;	(* set length of permanent data module		*)

			REPEAT	(* repeat until data of permanent memory data module have been read *)
				DatObjRead_01();						(* FUB read data from permanent data module 		*)
				UNTIL	DatObjRead_01.status <> ERR_FUB_BUSY		(* wait if FUB is busy 	*)
			END_REPEAT;

			IF DatObjRead_01.status <> ERR_NOERROR THEN	(* if status of read permanent data moduel is not OK 	*)
				pm_Error :=2012;						(* set permanent memory error status					*)
			END_IF
		END_IF;

		(* if permanent memory data module exist --> copy data from structure pm to program parameter *)
		IF pm_Error = ERR_NOERROR THEN

			(************ Permanent structure ************)
			(* ------------- V04.04.0 ---------------- *)		(* permanent memory data *)
			Para				:=	pmm;

		END_IF;
	END_IF

	(* create new permanent memory data module	*)
	IF bCreateDataObj THEN

		(* try to delete old data module *)
		DatObjDelete_PermMem.enable := TRUE;
		DatObjDelete_PermMem.ident 	:= pm_id;

		REPEAT	(* repeat until delete of permanent memory data module is ready *)
			DatObjDelete_PermMem();		(* FUB for delete permanent memory data module *)
			UNTIL	DatObjDelete_PermMem.status <> ERR_FUB_BUSY		(* wait if FUB is busy 	*)
		END_REPEAT;

		(* create new one *)
		DatObjCreate_01.enable	 := TRUE;			(* enable create permanent memory data module FUB 	*)
		DatObjCreate_01.grp 	 := 0;				(* must to be set to zero							*)
		DatObjCreate_01.pName 	 := ADR(ModulName);	(* set permanent memory data module name 			*)
		DatObjCreate_01.len 	 := pm_len;			(* set length ofpermanent memory data module		*)
		DatObjCreate_01.MemType  := doUSRROM;		(* create permanent memory data module at USERROM	*)
		DatObjCreate_01.Option 	 := 0;				(* cyclic checksum monitoring is on					*)
		DatObjCreate_01.pCpyData := 0;				(* no data will be copied do the permanent memory data module *)

		pm_Error:= 2003;							(* set permanent memory error status	*)

		REPEAT	(* repeat until generation of permanent memory data module is ready *)
			DatObjCreate_01();						(* FUB for create permanent memory data module 		*)
			UNTIL	DatObjCreate_01.status <> ERR_FUB_BUSY		(* wait if FUB is busy 	*)
		END_REPEAT;

		IF DatObjCreate_01.status = ERR_NOERROR THEN	(* is creation of permanent memory data module OK 	*)
			pm_p 	:= DatObjCreate_01.pDatObjMem;		(* set memory adress of permanent memory data module*)
			pm_id 	:= DatObjCreate_01.ident;			(* set identifier of permanent memory data module 	*)
		ELSE
			pm_Error:= 2004;							(* set permanent memory error status	*)
		END_IF;
	END_IF;

	(* prepare parameter for permanent memory data write in cyclic task *)
	IF pm_Error < 2004 THEN							(* permanent memory data module exist or has been created	*)
		DatObjWrite_01.enable 	:= TRUE;			(* enable permanent memory data module read FUB 	*)
		DatObjWrite_01.ident 	:= pm_id;			(* set identifier of permanent memory data module 	*)
		DatObjWrite_01.Offset 	:= 0;				(* start at memory offest zero 						*)
		DatObjWrite_01.pSource 	:= ADR(pmm);			(* set permanent memory data module name 			*)
		DatObjWrite_01.len 		:= pm_len;			(* set length ofpermanent memory data module		*)
	END_IF;

	(* calcualte actual checksum of parameter structure	*)
	ulChecksumOld := 0;			(* reset checksum value *)

	FOR ulPMPointer := ADR(pmm) TO (ADR(pmm) + pm_len - SIZEOF(ulChkValue)) DO
		memcpy(ADR(ulChkValue), ulPMPointer, SIZEOF(ulChkValue));
		ulChecksumOld := ulChecksumOld XOR ulChkValue;
	END_FOR;

END_PROGRAM
```

#### PermDI.var - Local variables
```iecst
VAR
	pm_Error : UINT;
	write_once : BOOL;
	pm_len : UDINT;
	ModulName : STRING[35];
	DatObjInfo_01 : DatObjInfo;
	pm_id : UDINT;
	pm_p : UDINT;
	bCreateDataObj : BOOL;
	perm_par_vers : UINT;
	DatObjRead_01 : DatObjRead;
	DatObjDelete_PermMem : DatObjDelete;
	DatObjCreate_01 : DatObjCreate;
	DatObjWrite_01 : DatObjWrite;
	ulChecksumOld : UDINT;
	ulPMPointer : UDINT;
	ulChkValue : UDINT;
	TON_WritePMEM : TON;
	ulChecksum : UDINT;
	bWriteDataObj : BOOL;
	TON_BlockMinFileAge : TON; (*waiting time without file write after successful performed write*)
	bBlock_MinFileAge : BOOL := FALSE; (*pause the perm file write after each sucessful write*)
	iPM_WriteCnt : UDINT; (* *) (*old VarName: usPMWriteCnt*)
END_VAR
VAR CONSTANT
	ERR_NOERROR : UINT := 0;
END_VAR
VAR
	pmm : Perm_DI_struct;
END_VAR
```

### Program Logical/DataInterface/VIS2PermDI (IEC, version 4.04.0) - + PermanentMemory

#### VIS2PermDICyclic.st - Cyclic code
```iecst
(*******************************************************************************
AGGR: read and write DIA.NE XT parameter to flash memory	(Cyclic)

This code is confidential and proprietary to the INNIO Jenbacher Company.
It may not be used in any form, or reproduced in any manner, without the express
written permission of the INNIO Company.
Copyright, INNIO Jenbacher Company, 2022

- every 10 seconds or at write once the parameter values are copied to the structure pm
- every 10 seconds the checksum of the parameter structure is calculate
- IF checksum has changed or write once is set the structure pm is written to
	the permanent memory data module

Customized modifications: -
------------------------

History:
-------
V1.00.0	16.09.2022	Vockenberger 	Neu erstellt
V1.03.0	22.01.2025	Gruber St.		added rCustEng2TB

*******************************************************************************)
PROGRAM _CYCLIC

	(* 10 seconds timer *)
	TON_WritePMEM(IN := NOT TON_WritePMEM.Q, PT:= T#10s);
	TON_BlockMinFileAge(IN := bBlock_MinFileAge, PT:= T#10m);
	IF TON_BlockMinFileAge.Q  THEN bBlock_MinFileAge := FALSE; END_IF

	(* every 10 seconds or at write once the parameter values are copied to the structure pm *)
	IF TON_WritePMEM.Q OR write_once THEN

		(* ------------- V04.04.0 ---------------- *)   					(* permanent memory data *)
		VIS2pmm.rFC_ChCW_LT_PuSet		:=	VIS2MM.rFC_ChCW_LT_PuSet;
		VIS2pmm.rFC_ChCW_HT_PuSet		:=	VIS2MM.rFC_ChCW_HT_PuSet;
		VIS2pmm.rFC_ChCW_LT_LP_PuSet	:=	VIS2MM.rFC_ChCW_LT_LP_PuSet;
		VIS2pmm.rFC_ChCW_LT_HP_PuSet	:=	VIS2MM.rFC_ChCW_LT_HP_PuSet;
		VIS2pmm.rFC_ChCW_HT_LP_PuSet	:=	VIS2MM.rFC_ChCW_HT_LP_PuSet;
		VIS2pmm.rFC_ChCW_HT_HP_PuSet	:=	VIS2MM.rFC_ChCW_HT_HP_PuSet;
		VIS2pmm.rFC_ECW_PuSet			:=	VIS2MM.rFC_ECW_PuSet;
		VIS2pmm.rFC_OCW_PuSet			:=	VIS2MM.rFC_OCW_PuSet;
		VIS2pmm.rCtr_RW_CV_Set			:=	VIS2MM.rCtr_RW_CV_Set;
		VIS2pmm.rCtr_RW_HE_Set			:=	VIS2MM.rCtr_RW_HE_Set;
		VIS2pmm.rCtr_RW_LT_1_Set		:=	VIS2MM.rCtr_RW_LT_1_Set;
		VIS2pmm.rCtr_RW_HT_1_Set		:=	VIS2MM.rCtr_RW_HT_1_Set;
		VIS2pmm.rCtr_RW_LT_2_Set		:=	VIS2MM.rCtr_RW_LT_2_Set;
		VIS2pmm.rCtr_RW_HT_2_Set		:=	VIS2MM.rCtr_RW_HT_2_Set;
		VIS2pmm.rCtr_RW_ECW_1_Set		:=	VIS2MM.rCtr_RW_ECW_1_Set;
		VIS2pmm.rCtr_RW_OCW_1_Set		:=	VIS2MM.rCtr_RW_OCW_1_Set;
		VIS2pmm.rCtr_RW_ECW_2_Set		:=	VIS2MM.rCtr_RW_ECW_2_Set;
		VIS2pmm.rCtr_RW_OCW_2_Set		:=	VIS2MM.rCtr_RW_OCW_2_Set;
		VIS2pmm.rMan_SRC_ByFlap_Set		:=	VIS2MM.rMan_SRC_ByFlap_Set;
		VIS2pmm.bECW_PreH_Dem_Customized := VIS2MM.bECW_PreH_Dem_Customized;
		VIS2pmm.rCtr_ChCW_LT_In_Y_set 	:=	VIS2MM.tCtr_ChCW_LT_In.Y_set;
		VIS2pmm.rCtr_ChCW_HT_In_Y_set 	:=	VIS2MM.tCtr_ChCW_HT_In.Y_set;
		VIS2pmm.rCtr_ChCW_LT_In_Y_set 	:=	VIS2MM.tCtr_ChCW_LT_In.Y_set;
		VIS2pmm.rCtr_ChCW_LT_In_Y_set 	:=	VIS2MM.tCtr_ChCW_LT_In.Y_set;
		VIS2pmm.rCtr_ChCW_HT_In_Y_set 	:=	VIS2MM.tCtr_ChCW_HT_In.Y_set;
		VIS2pmm.rCtr_ChCW_HT_In_Y_set 	:=	VIS2MM.tCtr_ChCW_HT_In.Y_set;
		VIS2pmm.rCtr_ECW_In_Y_set 		:=	VIS2MM.tCtr_ECW_In.Y_set;
		VIS2pmm.rCtr_OCW_In_Y_set 		:=	VIS2MM.tCtr_OCW_In.Y_set;
		VIS2pmm.bCtr_ChCW_LT_In_Y_set_Active := VIS2MM.tCtr_ChCW_LT_In.Y_set_Active;
		VIS2pmm.bCtr_ChCW_HT_In_Y_set_Active := VIS2MM.tCtr_ChCW_HT_In.Y_set_Active;
		VIS2pmm.bCtr_ChCW_LT_LP_In_Y_set_Active := VIS2MM.tCtr_ChCW_LT_LP_In.Y_set_Active;
		VIS2pmm.bCtr_ChCW_LT_HP_In_Y_set_Active := VIS2MM.tCtr_ChCW_LT_HP_In.Y_set_Active;
		VIS2pmm.bCtr_ChCW_HT_LP_In_Y_set_Active := VIS2MM.tCtr_ChCW_HT_LP_In.Y_set_Active;
		VIS2pmm.bCtr_ChCW_HT_HP_In_Y_set_Active := VIS2MM.tCtr_ChCW_HT_HP_In.Y_set_Active;
		VIS2pmm.bCtr_ECW_In_Y_set_Active 	:= VIS2MM.tCtr_ECW_In.Y_set_Active;
		VIS2pmm.bCtr_OCW_In_Y_set_Active 	:= VIS2MM.tCtr_OCW_In.Y_set_Active;
		VIS2pmm.bDem_ERV_Aut_Vis			:= VIS2MM.bDem_ERV_Aut_Vis;
		VIS2pmm.rMan_EG_Flap_Set			:= VIS2MM.rMan_EG_Flap_Set;
		VIS2pmm.rCust_Eng2TB				:= VIS2MM.rCust_Eng2TB;
		VIS2pmm.tPreHeatWDayLT				:= VIS2MM.tPreHeatWDayLT;
		VIS2pmm.bPreHeatWDayLT_CtrActive	:= VIS2MM.bPreHeatWDayLT_CtrActive;
		VIS2pmm.bLT_PreH_Dem				:= VIS2MM.bLT_PreH_Dem;
		VIS2pmm.rT_LT_HP_Preh				:= VIS2MM.rT_LT_HP_Preh;
		VIS2pmm.rT_LT_LP_Preh				:= VIS2MM.rT_LT_LP_Preh;
		VIS2pmm.bSel_PG_Comp				:= VIS2MM.bSel_PG_Comp;
		VIS2pmm.bSel_PG_TraceHeat			:= VIS2MM.bSel_PG_TraceHeat;
		VIS2pmm.bSel_PG_TraceHeat_TimeCtr	:= VIS2MM.bSel_PG_TraceHeat_TimeCtr;
		VIS2pmm.rCtr_PG_CompSet				:= VIS2MM.rCtr_PG_CompSet;
		VIS2pmm.rOp_ExhFlap					:= VIS2MM.rOp_ExhFlap;
		VIS2pmm.bCool_Air_Active			:= VIS2MM.bCool_Air_Active;
	END_IF;

	(* cyclic calcualtion of parameter checksum	*)
	IF TON_WritePMEM.Q THEN
		ulChecksum := 0;

		FOR ulPMPointer := ADR(VIS2pmm) TO (ADR(VIS2pmm) + pm_len - SIZEOF(ulChkValue)) DO
			memcpy(ADR(ulChkValue), ulPMPointer, SIZEOF(ulChkValue));
			ulChecksum := (ulChecksum XOR ulChkValue)+ulChkValue;
		END_FOR;

		IF ulChecksumOld <> ulChecksum THEN	(* if checksum has changed 		*)
			ulChecksumOld := ulChecksum;	(* save last cheksum value		*)
			bWriteDataObj := TRUE;			(* set flag for write checksum	*)
		END_IF;

	END_IF

	(* write structure pm to the permanent memory module *)
	IF ((bWriteDataObj AND NOT bBlock_MinFileAge) OR write_once) THEN

		DatObjWrite_01();									(* run data object write fub 				*)

		IF DatObjWrite_01.status <> ERR_FUB_BUSY THEN		(* wait if data object write fub is busy 	*)
			bWriteDataObj 	:= FALSE;						(* reset data object write flag				*)
			write_once 		:= FALSE;						(* reset write_once flag 					*)
			iPM_WriteCnt 	:= iPM_WriteCnt + 1;			(* counter for done data object module writes *)

			IF DatObjWrite_01.status = ERR_NOERROR THEN		(* if status = NO ERROR -> block further write requests for 10min to avoid CF wear down	*)
				bBlock_MinFileAge := TRUE;
			ELSE
				pm_Error := 2005;							(* set data object write error state		*)
			END_IF;
		END_IF;

	END_IF;

END_PROGRAM
```

#### VIS2PermDIInit.st - Initialization code
```iecst
(*******************************************************************************
AGGR: read and write DIA.NE XT parameter to flash memory	(init)

This code is confidential and proprietary to the INNIO Jenbacher Company.
It may not be used in any form, or reproduced in any manner, without the express
written permission of the INNIO Company.
Copyright, INNIO Jenbacher Company, 2022

- every 10 seconds or at write once the parameter values are copied to the structure pm
- every 10 seconds the checksum of the parameter structure is calculate
- IF checksum has changed or write once is set the structure pm is written to
	the permanent memory data module

Customized modifications: -
------------------------

History:
-------
V1.00.0	16.09.2022	Vockenberger 	Neu erstellt
V1.03.0	22.01.2025	Gruber St.		added rCustEng2TB

*******************************************************************************)

PROGRAM _INIT

	(* set some init parameters *)
	TON_WritePMEM(IN := FALSE, PT:= T#10s);			(* reset used timer function blocks 			*)

	pm_Error 	:= ERR_NOERROR;						(* reset permanent memory error	status			*)
	write_once 	:= FALSE;				 			(* reset flag for write permanent memory once	*)
	pm_len 		:= SIZEOF(VIS2pmm);						(* define data length of permenent memory		*)
	strcpy(ADR(ModulName),ADR('DataInterface::VISpm_DI'));	(* define name of permanent memory data module	*)

	(* check for existing permanent memory data module	*)
	DatObjInfo_01.enable:= TRUE;					(* enable FUB									*)
	DatObjInfo_01.pName := ADR(ModulName);			(* set permanent memory data module name 		*)
	DatObjInfo_01();								(* run data object info FUB						*)

	(* check error status of data object info FUB	*)
	IF DatObjInfo_01.status = ERR_NOERROR THEN		(* if no error	--> permanent memory data module exists	*)
		pm_id 	:= DatObjInfo_01.ident;				(* copy permanent memory data module ident			*)
		pm_p 	:= DatObjInfo_01.pDatObjMem;		(* copy permanent memory data module memory adres	*)
	ELSE
		bCreateDataObj := TRUE;						(* set flag for create new data object	*)
		pm_Error := 2001;							(* set permanent memory error status	*)
	END_IF;

	(* check length of parameter struct with length of data object *)

	CASE DatObjInfo_01.len OF

		456: 		perm_par_vers  := 400;			(* 44 = length of perm_par V04.00.0 *)

			(* insert new perm_par Version here
			(* 		  bCreateDataObj := TRUE;		(* set flag for create new data object	*)
			(* xxxx:  perm_par_vers  := yyy;		(* xxxx = length of perm_par Vy.yy *)

		ELSE
		bCreateDataObj := TRUE;						(* set flag for create new data object	*)
	END_CASE;

	(* if permanent memory data module exist read data and copy to structure pm	*)
	IF pm_Error = ERR_NOERROR THEN					(* permanent memory data module exist 				*)
		DatObjRead_01.enable 		:= TRUE;		(* enable read permanent memory module data 		*)
		DatObjRead_01.ident 		:= pm_id;		(* set identifier of permanent memory data module	*)
		DatObjRead_01.Offset 		:= 0;			(* start at memory offest zero 						*)
		DatObjRead_01.pDestination := ADR(VIS2pmm);		(* set permanent data destination adress			*)
		DatObjRead_01.len 			:= DatObjInfo_01.len;	(* set length of permanent data module		*)

		REPEAT	(* repeat until data of permanent memory data module have been read *)
			DatObjRead_01();						(* FUB read data from permanent data module 		*)
			UNTIL	DatObjRead_01.status <> ERR_FUB_BUSY		(* wait if FUB is busy 	*)
		END_REPEAT;

		IF DatObjRead_01.status <> ERR_NOERROR THEN	(* if status of read permanent data moduel is not OK 	*)
			pm_Error :=2002;						(* set permanent memory error status					*)
		END_IF
	END_IF;

	IF NOT bCreateDataObj THEN
		(* if permanent memory data module exist read data and copy to structure pm	*)
		IF pm_Error = ERR_NOERROR THEN					(* permanent memory data module exist 				*)
			DatObjRead_01.enable 		:= TRUE;		(* enable read permanent memory module data 		*)
			DatObjRead_01.ident 		:= pm_id;		(* set identifier of permanent memory data module	*)
			DatObjRead_01.Offset 		:= 0;			(* start at memory offest zero 						*)
			DatObjRead_01.pDestination := ADR(VIS2pmm);		(* set permanent data destination adress			*)
			DatObjRead_01.len 			:= DatObjInfo_01.len;	(* set length of permanent data module		*)

			REPEAT	(* repeat until data of permanent memory data module have been read *)
				DatObjRead_01();						(* FUB read data from permanent data module 		*)
				UNTIL	DatObjRead_01.status <> ERR_FUB_BUSY		(* wait if FUB is busy 	*)
			END_REPEAT;

			IF DatObjRead_01.status <> ERR_NOERROR THEN	(* if status of read permanent data moduel is not OK 	*)
				pm_Error :=2012;						(* set permanent memory error status					*)
			END_IF
		END_IF;

		(* if permanent memory data module exist --> copy data from structure pm to program parameter *)
		IF pm_Error = ERR_NOERROR THEN

			(************ Permanent structure ************)
			(* ------------- V04.04.0 ---------------- *)		(* permanent memory data *)
			VIS2MM.rFC_ChCW_LT_PuSet		:=	VIS2pmm.rFC_ChCW_LT_PuSet;
			VIS2MM.rFC_ChCW_HT_PuSet		:=	VIS2pmm.rFC_ChCW_HT_PuSet;
			VIS2MM.rFC_ChCW_LT_LP_PuSet		:=	VIS2pmm.rFC_ChCW_LT_LP_PuSet;
			VIS2MM.rFC_ChCW_LT_HP_PuSet		:=	VIS2pmm.rFC_ChCW_LT_HP_PuSet;
			VIS2MM.rFC_ChCW_HT_LP_PuSet		:=	VIS2pmm.rFC_ChCW_HT_LP_PuSet;
			VIS2MM.rFC_ChCW_HT_HP_PuSet		:=	VIS2pmm.rFC_ChCW_HT_HP_PuSet;
			VIS2MM.rFC_ECW_PuSet			:=	VIS2pmm.rFC_ECW_PuSet;
			VIS2MM.rFC_OCW_PuSet			:=	VIS2pmm.rFC_OCW_PuSet;
			VIS2MM.rCtr_RW_CV_Set			:=	VIS2pmm.rCtr_RW_CV_Set;
			VIS2MM.rCtr_RW_HE_Set			:=	VIS2pmm.rCtr_RW_HE_Set;
			VIS2MM.rCtr_RW_LT_1_Set			:=	VIS2pmm.rCtr_RW_LT_1_Set;
			VIS2MM.rCtr_RW_HT_1_Set			:=	VIS2pmm.rCtr_RW_HT_1_Set;
			VIS2MM.rCtr_RW_LT_2_Set			:=	VIS2pmm.rCtr_RW_LT_2_Set;
			VIS2MM.rCtr_RW_HT_2_Set			:=	VIS2pmm.rCtr_RW_HT_2_Set;
			VIS2MM.rCtr_RW_ECW_1_Set		:=	VIS2pmm.rCtr_RW_ECW_1_Set;
			VIS2MM.rCtr_RW_OCW_1_Set		:=	VIS2pmm.rCtr_RW_OCW_1_Set;
			VIS2MM.rCtr_RW_ECW_2_Set		:=	VIS2pmm.rCtr_RW_ECW_2_Set;
			VIS2MM.rCtr_RW_OCW_2_Set		:=	VIS2pmm.rCtr_RW_OCW_2_Set;
			VIS2MM.rMan_SRC_ByFlap_Set		:=	VIS2pmm.rMan_SRC_ByFlap_Set;
			VIS2MM.bECW_PreH_Dem_Customized :=	VIS2pmm.bECW_PreH_Dem_Customized;
			VIS2MM.tCtr_ChCW_LT_In.Y_set 	:=	VIS2pmm.rCtr_ChCW_LT_In_Y_set;
			VIS2MM.tCtr_ChCW_HT_In.Y_set 	:=	VIS2pmm.rCtr_ChCW_HT_In_Y_set;
			VIS2MM.tCtr_ChCW_LT_In.Y_set 	:=	VIS2pmm.rCtr_ChCW_LT_In_Y_set;
			VIS2MM.tCtr_ChCW_LT_In.Y_set 	:=	VIS2pmm.rCtr_ChCW_LT_In_Y_set;
			VIS2MM.tCtr_ChCW_HT_In.Y_set 	:=	VIS2pmm.rCtr_ChCW_HT_In_Y_set;
			VIS2MM.tCtr_ChCW_HT_In.Y_set 	:=	VIS2pmm.rCtr_ChCW_HT_In_Y_set;
			VIS2MM.tCtr_ECW_In.Y_set 		:=	VIS2pmm.rCtr_ECW_In_Y_set;
			VIS2MM.tCtr_OCW_In.Y_set 		:=	VIS2pmm.rCtr_OCW_In_Y_set;
			VIS2MM.tCtr_ChCW_LT_In.Y_set_Active := VIS2pmm.bCtr_ChCW_LT_In_Y_set_Active;
			VIS2MM.tCtr_ChCW_HT_In.Y_set_Active := VIS2pmm.bCtr_ChCW_HT_In_Y_set_Active;
			VIS2MM.tCtr_ChCW_LT_LP_In.Y_set_Active := VIS2pmm.bCtr_ChCW_LT_LP_In_Y_set_Active;
			VIS2MM.tCtr_ChCW_LT_HP_In.Y_set_Active := VIS2pmm.bCtr_ChCW_LT_HP_In_Y_set_Active;
			VIS2MM.tCtr_ChCW_HT_LP_In.Y_set_Active := VIS2pmm.bCtr_ChCW_HT_LP_In_Y_set_Active;
			VIS2MM.tCtr_ChCW_HT_HP_In.Y_set_Active := VIS2pmm.bCtr_ChCW_HT_HP_In_Y_set_Active;
			VIS2MM.tCtr_ECW_In.Y_set_Active 	:= VIS2pmm.bCtr_ECW_In_Y_set_Active;
			VIS2MM.tCtr_OCW_In.Y_set_Active 	:= VIS2pmm.bCtr_OCW_In_Y_set_Active;
			VIS2MM.bDem_ERV_Aut_Vis				:= VIS2pmm.bDem_ERV_Aut_Vis;
			VIS2MM.rMan_EG_Flap_Set				:= VIS2pmm.rMan_EG_Flap_Set;
			VIS2MM.rCust_Eng2TB					:= VIS2pmm.rCust_Eng2TB;
			VIS2MM.tPreHeatWDayLT				:= VIS2pmm.tPreHeatWDayLT;
			VIS2MM.bPreHeatWDayLT_CtrActive		:= VIS2pmm.bPreHeatWDayLT_CtrActive;
			VIS2MM.bLT_PreH_Dem					:= VIS2pmm.bLT_PreH_Dem;
			VIS2MM.rT_LT_HP_Preh				:= VIS2pmm.rT_LT_HP_Preh;
			VIS2MM.rT_LT_LP_Preh				:= VIS2pmm.rT_LT_LP_Preh;
			VIS2MM.bSel_PG_Comp					:= VIS2pmm.bSel_PG_Comp;
			VIS2MM.bSel_PG_TraceHeat			:= VIS2pmm.bSel_PG_TraceHeat;
			VIS2MM.bSel_PG_TraceHeat_TimeCtr	:= VIS2pmm.bSel_PG_TraceHeat_TimeCtr;
			VIS2MM.rCtr_PG_CompSet				:= VIS2pmm.rCtr_PG_CompSet;
			VIS2MM.rOp_ExhFlap					:= VIS2pmm.rOp_ExhFlap;
			VIS2MM.bCool_Air_Active				:= VIS2pmm.bCool_Air_Active;
		END_IF;
	END_IF

	(* create new permanent memory data module	*)
	IF bCreateDataObj THEN

		(* try to delete old data module *)
		DatObjDelete_PermMem.enable := TRUE;
		DatObjDelete_PermMem.ident 	:= pm_id;

		REPEAT	(* repeat until delete of permanent memory data module is ready *)
			DatObjDelete_PermMem();		(* FUB for delete permanent memory data module *)
			UNTIL	DatObjDelete_PermMem.status <> ERR_FUB_BUSY		(* wait if FUB is busy 	*)
		END_REPEAT;

		(* create new one *)
		DatObjCreate_01.enable	 := TRUE;			(* enable create permanent memory data module FUB 	*)
		DatObjCreate_01.grp 	 := 0;				(* must to be set to zero							*)
		DatObjCreate_01.pName 	 := ADR(ModulName);	(* set permanent memory data module name 			*)
		DatObjCreate_01.len 	 := pm_len;			(* set length ofpermanent memory data module		*)
		DatObjCreate_01.MemType  := doUSRROM;		(* create permanent memory data module at USERROM	*)
		DatObjCreate_01.Option 	 := 0;				(* cyclic checksum monitoring is on					*)
		DatObjCreate_01.pCpyData := 0;				(* no data will be copied do the permanent memory data module *)

		pm_Error:= 2003;							(* set permanent memory error status	*)

		REPEAT	(* repeat until generation of permanent memory data module is ready *)
			DatObjCreate_01();						(* FUB for create permanent memory data module 		*)
			UNTIL	DatObjCreate_01.status <> ERR_FUB_BUSY		(* wait if FUB is busy 	*)
		END_REPEAT;

		IF DatObjCreate_01.status = ERR_NOERROR THEN	(* is creation of permanent memory data module OK 	*)
			pm_p 	:= DatObjCreate_01.pDatObjMem;		(* set memory adress of permanent memory data module*)
			pm_id 	:= DatObjCreate_01.ident;			(* set identifier of permanent memory data module 	*)
		ELSE
			pm_Error:= 2004;							(* set permanent memory error status	*)
		END_IF;
	END_IF;

	(* prepare parameter for permanent memory data write in cyclic task *)
	IF pm_Error < 2004 THEN							(* permanent memory data module exist or has been created	*)
		DatObjWrite_01.enable 	:= TRUE;			(* enable permanent memory data module read FUB 	*)
		DatObjWrite_01.ident 	:= pm_id;			(* set identifier of permanent memory data module 	*)
		DatObjWrite_01.Offset 	:= 0;				(* start at memory offest zero 						*)
		DatObjWrite_01.pSource 	:= ADR(VIS2pmm);			(* set permanent memory data module name 			*)
		DatObjWrite_01.len 		:= pm_len;			(* set length ofpermanent memory data module		*)
	END_IF;

	(* calcualte actual checksum of parameter structure	*)
	ulChecksumOld := 0;			(* reset checksum value *)

	FOR ulPMPointer := ADR(VIS2pmm) TO (ADR(VIS2pmm) + pm_len - SIZEOF(ulChkValue)) DO
		memcpy(ADR(ulChkValue), ulPMPointer, SIZEOF(ulChkValue));
		ulChecksumOld := ulChecksumOld XOR ulChkValue;
	END_FOR;

END_PROGRAM
```

#### VIS2PermDI.var - Local variables
```iecst
VAR
	pm_Error : UINT;
	write_once : BOOL;
	pm_len : UDINT;
	ModulName : STRING[35];
	DatObjInfo_01 : DatObjInfo;
	pm_id : UDINT;
	pm_p : UDINT;
	bCreateDataObj : BOOL;
	perm_par_vers : UINT;
	DatObjRead_01 : DatObjRead;
	DatObjDelete_PermMem : DatObjDelete;
	DatObjCreate_01 : DatObjCreate;
	DatObjWrite_01 : DatObjWrite;
	ulChecksumOld : UDINT;
	ulPMPointer : UDINT;
	ulChkValue : UDINT;
	TON_WritePMEM : TON;
	ulChecksum : UDINT;
	bWriteDataObj : BOOL;
	TON_BlockMinFileAge : TON; (*waiting time without file write after successful performed write*)
	bBlock_MinFileAge : BOOL := FALSE; (*pause the perm file write after each sucessful write*)
	iPM_WriteCnt : UDINT; (* *) (*old VarName: usPMWriteCnt*)
END_VAR
VAR CONSTANT
	ERR_NOERROR : UINT := 0;
END_VAR
VAR
	VIS2pmm : VIS2perm_DI_struct;
END_VAR
```

Listed in the project but not available here: Logical/Libraries/MATLAB_includes/R2012b/rtw_solver.h, Logical/Libraries/MATLAB_includes/R2012b/rtw_windows.h, Logical/Libraries/MATLAB_includes/R2012b/rtw_xpc.h, Logical/Libraries/MATLAB_includes/R2012b/sfcn_bridge.h, Logical/Libraries/MATLAB_includes/R2012b/sfun_rtwcg.hpp, Logical/Libraries/MATLAB_includes/R2012b/sigmapdef_sfcn.h, Logical/Libraries/MATLAB_includes/R2012b/sigregdef.h, Logical/Libraries/MATLAB_includes/R2012b/simstruc.h, Logical/Libraries/MATLAB_includes/R2012b/simstruc_types.h, Logical/Libraries/MATLAB_includes/R2012b/simulink.h, Logical/Libraries/MATLAB_includes/R2012b/simulink2.h, Logical/Libraries/MATLAB_includes/R2012b/simulink_solver_api.h, Logical/Libraries/MATLAB_includes/R2012b/sl_common_types_def.h, Logical/Libraries/MATLAB_includes/R2012b/sl_datatype_access.h, Logical/Libraries/MATLAB_includes/R2012b/sl_fileio_rtw.h, Logical/Libraries/MATLAB_includes/R2012b/sl_fixpt.h, Logical/Libraries/MATLAB_includes/R2012b/sl_prodhwdevicetype.h, Logical/Libraries/MATLAB_includes/R2012b/sl_sample_time_defs.h, Logical/Libraries/MATLAB_includes/R2012b/sl_solver_rtw.h, Logical/Libraries/MATLAB_includes/R2012b/sl_types_def.h, Logical/Libraries/MATLAB_includes/R2012b/slexec_ssbridge.h, Logical/Libraries/MATLAB_includes/R2012b/solver_zc.h, Logical/Libraries/MATLAB_includes/R2012b/sysran_types.h, Logical/Libraries/MATLAB_includes/R2012b/tmwtypes.h, Logical/Libraries/MATLAB_includes/R2012b/updown.h, Logical/Libraries/MATLAB_includes/R2012b/updown_util.h, Logical/Libraries/MATLAB_includes/R2012b/upsup_public.h, Logical/Libraries/MATLAB_includes/R2020a, Logical/Libraries/MATLAB_includes/R2021b, Logical/Monic/CAN/caniniMo, Logical/Monic/CAN/cmsmonic, Logical/SAFI/DataSA/sa_coil, Logical/SAFI/DataSA/sa_curr, Logical/SAFI/CAN/Updater, Logical/SAFI/CAN/canmaiSA, Logical/SAFI/CAN/caniniSA, Logical/SAFI/CAN/sadmr24, Logical/SAFI/CAN/sagen24, Logical/SAFI/CAN/saign24, Logical/SAFI/CAN/sakls24, Logical/SAFI/CAN/sapi24, Logical/SAFI/CAN/sadmr1_12, Logical/SAFI/CAN/sagen1_12, Logical/SAFI/CAN/saign1_12, Logical/SAFI/CAN/sakls1_12, Logical/SAFI/CAN/sapi1_12, Logical/SAFI/CAN/sadmr13_24, Logical/SAFI/CAN/sagen13_24, Logical/SAFI/CAN/saign13_24, Logical/SAFI/CAN/sakls13_24, Logical/SAFI/CAN/sapi13_24, Logical/SAFI/CAN/sadmr1_10, Logical/SAFI/CAN/sagen1_10, Logical/SAFI/CAN/saign1_10, Logical/SAFI/CAN/sakls1_10, Logical/SAFI/CAN/sapi1_10, Logical/SAFI/CAN/sadmr11_20, Logical/SAFI/CAN/sagen11_20, Logical/SAFI/CAN/saign11_20, Logical/SAFI/CAN/sakls11_20, Logical/SAFI/CAN/sapi11_20, Logical/SAFI/CAN/sadmr1_8, Logical/SAFI/CAN/sagen1_8, Logical/SAFI/CAN/saign1_8, Logical/SAFI/CAN/sakls1_8, Logical/SAFI/CAN/sapi1_8, Logical/SAFI/CAN/sadmr9_16, Logical/SAFI/CAN/sagen9_16, Logical/SAFI/CAN/saign9_16, Logical/SAFI/CAN/sakls9_16, Logical/SAFI/CAN/sapi9_16, Logical/SAFI/CAN/sadmr1_6, Logical/SAFI/CAN/sagen1_6, Logical/SAFI/CAN/saign1_6, Logical/SAFI/CAN/sakls1_6, Logical/SAFI/CAN/sapi1_6, Logical/SAFI/CAN/sadmr7_12, Logical/SAFI/CAN/sagen7_12, Logical/SAFI/CAN/saign7_12, Logical/SAFI/CAN/sakls7_12, Logical/SAFI/CAN/sapi7_12
